LIN {X 0,Y 183.152,Z 369.76,A -85,B 0,C 180,E1 -22263.807,E2 -22263.807} C_VEL
LIN {X 0,Y 182.882,Z 372.565,A -85,B 0,C 180,E1 -22267.944,E2 -22267.944} C_VEL
LIN {X 0,Y 183.104,Z 373.609,A -85,B 0,C 180,E1 -22270.732,E2 -22270.732} C_VEL
LIN {X 0,Y 183.564,Z 374.058,A -85,B 0,C 180,E1 -22273.565,E2 -22273.565} C_VEL
LIN {X 0,Y 184.444,Z 373.742,A -85,B 0,C 180,E1 -22276.698,E2 -22276.698} C_VEL
LIN {X 0,Y 185.786,Z 372.532,A -85,B 0,C 180,E1 -22279.98,E2 -22279.98} C_VEL
LIN {X 0,Y 187.578,Z 370.431,A -85,B 0,C 180,E1 -22283.169,E2 -22283.169} C_VEL
LIN {X 0,Y 189.778,Z 367.45,A -85,B 0,C 180,E1 -22286.257,E2 -22286.257} C_VEL
LIN {X 0,Y 193.019,Z 362.657,A -85,B 0,C 180,E1 -22289.797,E2 -22289.797} C_VEL
LIN {X 0,Y 196.874,Z 356.364,A -85,B 0,C 180,E1 -22293.185,E2 -22293.185} C_VEL
LIN {X 0,Y 200.364,Z 350.078,A -85,B 0,C 180,E1 -22295.784,E2 -22295.784} C_VEL
LIN {X 0,Y 204.762,Z 341.315,A -85,B 0,C 180,E1 -22298.595,E2 -22298.595} C_VEL
LIN {X 0,Y 209.064,Z 331.687,A -85,B 0,C 180,E1 -22300.994,E2 -22300.994} C_VEL
LIN {X 0,Y 213.104,Z 321.145,A -85,B 0,C 180,E1 -22303.022,E2 -22303.022} C_VEL
LIN {X 0,Y 216.763,Z 309.855,A -85,B 0,C 180,E1 -22304.707,E2 -22304.707} C_VEL
LIN {X 0,Y 219.632,Z 298.789,A -85,B 0,C 180,E1 -22305.997,E2 -22305.997} C_VEL
LIN {X 0,Y 222.031,Z 286.626,A -85,B 0,C 180,E1 -22307.061,E2 -22307.061} C_VEL
LIN {X 0,Y 223.839,Z 274.15,A -85,B 0,C 180,E1 -22307.808,E2 -22307.808} C_VEL
LIN {X 0,Y 226.368,Z 244.862,A -85,B 0,C 180,E1 -22308.842,E2 -22308.842} C_VEL
LIN {X 0,Y 227.604,Z 229.196,A -85,B 0,C 180,E1 -22309.377,E2 -22309.377} C_VEL
LIN {X 0,Y 223.853,Z 221.057,A -85,B 0,C 180,E1 -22311.183,E2 -22311.183} C_VEL
LIN {X 0,Y 219.292,Z 213.106,A -85,B 0,C 180,E1 -22313.476,E2 -22313.476} C_VEL
LIN {X 0,Y 214.6,Z 205.629,A -85,B 0,C 180,E1 -22316.16,E2 -22316.16} C_VEL
LIN {X 0,Y 212.303,Z 202.347,A -85,B 0,C 180,E1 -22317.592,E2 -22317.592} C_VEL
LIN {X 0,Y 209.697,Z 198.642,A -85,B 0,C 180,E1 -22319.412,E2 -22319.412} C_VEL
LIN {X 0,Y 208.666,Z 197.162,A -85,B 0,C 180,E1 -22320.182,E2 -22320.182} C_VEL
LIN {X 0,Y 206.119,Z 193.314,A -85,B 0,C 180,E1 -22322.322,E2 -22322.322} C_VEL
LIN {X 0,Y 203.232,Z 190.633,A -85,B 0,C 180,E1 -22324.977,E2 -22324.977} C_VEL
LIN {X 0,Y 202.029,Z 188.256,A -85,B 0,C 180,E1 -22326.493,E2 -22326.493} C_VEL
LIN {X 0,Y 198.406,Z 185.102,A -85,B 0,C 180,E1 -22332.017,E2 -22332.017} C_VEL
LIN {X 0,Y 197.661,Z 183.274,A -85,B 0,C 180,E1 -22334.413,E2 -22334.413} C_VEL
LIN {X 0,Y 196.972,Z 183.268,A -85,B 0,C 180,E1 -22338.732,E2 -22338.732} C_VEL
LIN {X 0,Y 198.03,Z 184.97,A -85,B 0,C 180,E1 -22344.495,E2 -22344.495} C_VEL
LIN {X 0,Y 198.934,Z 186.56,A -85,B 0,C 180,E1 -22346.631,E2 -22346.631} C_VEL
LIN {X 0,Y 203.525,Z 193.122,A -85,B 0,C 180,E1 -22352.933,E2 -22352.933} C_VEL
LIN {X 0,Y 206.778,Z 198.314,A -85,B 0,C 180,E1 -22356.036,E2 -22356.036} C_VEL
LIN {X 0,Y 211.278,Z 205.799,A -85,B 0,C 180,E1 -22359.489,E2 -22359.489} C_VEL
LIN {X 0,Y 214.488,Z 211.478,A -85,B 0,C 180,E1 -22361.581,E2 -22361.581} C_VEL
LIN {X 0,Y 217.853,Z 217.949,A -85,B 0,C 180,E1 -22363.597,E2 -22363.597} C_VEL
LIN {X 0,Y 221.896,Z 226.386,A -85,B 0,C 180,E1 -22365.77,E2 -22365.77} C_VEL
LIN {X 0,Y 226.021,Z 237.025,A -85,B 0,C 180,E1 -22367.898,E2 -22367.898} C_VEL
LIN {X 0,Y 226.566,Z 244.834,A -85,B 0,C 180,E1 -22368.537,E2 -22368.537} C_VEL
LIN {X 0,Y 224.824,Z 267.129,A -85,B 0,C 180,E1 -22369.298,E2 -22369.298} C_VEL
LIN {X 0,Y 223.917,Z 272.973,A -85,B 0,C 180,E1 -22369.35,E2 -22369.35} C_VEL
LIN {X 0,Y 221.191,Z 282.484,A -85,B 0,C 180,E1 -22369.097,E2 -22369.097} C_VEL
LIN {X 0,Y 218.142,Z 291.897,A -85,B 0,C 180,E1 -22368.96,E2 -22368.96} C_VEL
LIN {X 0,Y 216.749,Z 297.576,A -85,B 0,C 180,E1 -22369.179,E2 -22369.179} C_VEL
LIN {X 0,Y 213.874,Z 310.256,A -85,B 0,C 180,E1 -22370.149,E2 -22370.149} C_VEL
LIN {X 0,Y 210.254,Z 322.7,A -85,B 0,C 180,E1 -22371.495,E2 -22371.495} C_VEL
LIN {X 0,Y 205.689,Z 335.169,A -85,B 0,C 180,E1 -22373.276,E2 -22373.276} C_VEL
LIN {X 0,Y 201.948,Z 344.09,A -85,B 0,C 180,E1 -22374.954,E2 -22374.954} C_VEL
LIN {X 0,Y 197.526,Z 353.357,A -85,B 0,C 180,E1 -22377.138,E2 -22377.138} C_VEL
LIN {X 0,Y 192.824,Z 362.381,A -85,B 0,C 180,E1 -22379.922,E2 -22379.922} C_VEL
LIN {X 0,Y 188.656,Z 369.747,A -85,B 0,C 180,E1 -22382.847,E2 -22382.847} C_VEL
LIN {X 0,Y 184.654,Z 376.594,A -85,B 0,C 180,E1 -22386.443,E2 -22386.443} C_VEL
LIN {X 0,Y 181.708,Z 381.181,A -85,B 0,C 180,E1 -22389.628,E2 -22389.628} C_VEL
LIN {X 0,Y 178.635,Z 385.659,A -85,B 0,C 180,E1 -22394.013,E2 -22394.013} C_VEL
LIN {X 0,Y 177.625,Z 387.289,A -85,B 0,C 180,E1 -22396.266,E2 -22396.266} C_VEL
LIN {X 0,Y 176.39,Z 389.3,A -85,B 0,C 180,E1 -22400.828,E2 -22400.828} C_VEL
LIN {X 0,Y 176.069,Z 389.772,A -85,B 0,C 180,E1 -22405.42,E2 -22405.42} C_VEL
LIN {X 0,Y 176.19,Z 389.418,A -85,B 0,C 180,E1 -22407.713,E2 -22407.713} C_VEL
LIN {X 0,Y 176.407,Z 388.626,A -85,B 0,C 180,E1 -22409.999,E2 -22409.999} C_VEL
LIN {X 0,Y 176.256,Z 387.392,A -85,B 0,C 180,E1 -22412.284,E2 -22412.284} C_VEL
LIN {X 0,Y 176.176,Z 384.702,A -85,B 0,C 180,E1 -22415.722,E2 -22415.722} C_VEL
LIN {X 0,Y 176.508,Z 380.942,A -85,B 0,C 180,E1 -22419.163,E2 -22419.163} C_VEL
LIN {X 0,Y 177.165,Z 375.989,A -85,B 0,C 180,E1 -22422.601,E2 -22422.601} C_VEL
LIN {X 0,Y 178.446,Z 369.723,A -85,B 0,C 180,E1 -22426.002,E2 -22426.002} C_VEL
LIN {X 0,Y 180.258,Z 361.863,A -85,B 0,C 180,E1 -22429.353,E2 -22429.353} C_VEL
LIN {X 0,Y 182.174,Z 353.728,A -85,B 0,C 180,E1 -22432.113,E2 -22432.113} C_VEL
LIN {X 0,Y 184.49,Z 343.939,A -85,B 0,C 180,E1 -22434.772,E2 -22434.772} C_VEL
LIN {X 0,Y 186.674,Z 334.322,A -85,B 0,C 180,E1 -22436.857,E2 -22436.857} C_VEL
LIN {X 0,Y 188.827,Z 324.044,A -85,B 0,C 180,E1 -22438.632,E2 -22438.632} C_VEL
LIN {X 0,Y 190.99,Z 311.886,A -85,B 0,C 180,E1 -22440.242,E2 -22440.242} C_VEL
LIN {X 0,Y 192.737,Z 299.331,A -85,B 0,C 180,E1 -22441.458,E2 -22441.458} C_VEL
LIN {X 0,Y 194.06,Z 286.706,A -85,B 0,C 180,E1 -22442.287,E2 -22442.287} C_VEL
LIN {X 0,Y 196.483,Z 238.495,A -85,B 0,C 180,E1 -22444.227,E2 -22444.227} C_VEL
LIN {X 0,Y 193.478,Z 211.936,A -85,B 0,C 180,E1 -22445.896,E2 -22445.896} C_VEL
LIN {X 0,Y 185.743,Z 191.175,A -85,B 0,C 180,E1 -22448.157,E2 -22448.157} C_VEL
LIN {X 0,Y 179.959,Z 177.42,A -85,B 0,C 180,E1 -22449.964,E2 -22449.964} C_VEL
LIN {X 0,Y 178.427,Z 171.263,A -85,B 0,C 180,E1 -22453.455,E2 -22453.455} C_VEL
LIN {X 0,Y 178.403,Z 171.26,A -85,B 0,C 180,E1 -22458.457,E2 -22458.457} C_VEL
LIN {X 0,Y 178.422,Z 171.263,A -85,B 0,C 180,E1 -22463.782,E2 -22463.782} C_VEL
LIN {X 0,Y 178.487,Z 171.252,A -85,B 0,C 180,E1 -22466.545,E2 -22466.545} C_VEL
LIN {X 0,Y 178.522,Z 171.241,A -85,B 0,C 180,E1 -22470.005,E2 -22470.005} C_VEL
LIN {X 0,Y 178.534,Z 171.244,A -85,B 0,C 180,E1 -22474.874,E2 -22474.874} C_VEL
LIN {X 0,Y 178.59,Z 171.24,A -85,B 0,C 180,E1 -22480.812,E2 -22480.812} C_VEL
LIN {X 0,Y 178.648,Z 171.23,A -85,B 0,C 180,E1 -22486.346,E2 -22486.346} C_VEL
LIN {X 0,Y 178.957,Z 171.183,A -85,B 0,C 180,E1 -22490.961,E2 -22490.961} C_VEL
LIN {X 0,Y 179.152,Z 171.167,A -85,B 0,C 180,E1 -22497.751,E2 -22497.751} C_VEL
LIN {X 0,Y 179.37,Z 171.135,A -85,B 0,C 180,E1 -22499.999,E2 -22499.999} C_VEL
LIN {X 0,Y 178.87,Z 171.194,A -85,B 0,C 180,E1 -22504.506,E2 -22504.506} C_VEL
LIN {X 0,Y 178.956,Z 171.192,A -85,B 0,C 180,E1 -22509.037,E2 -22509.037} C_VEL
LIN {X 0,Y 178.683,Z 171.207,A -85,B 0,C 180,E1 -22513.649,E2 -22513.649} C_VEL
LIN {X 0,Y 178.65,Z 171.229,A -85,B 0,C 180,E1 -22518.342,E2 -22518.342} C_VEL
LIN {X 0,Y 178.519,Z 171.237,A -85,B 0,C 180,E1 -22523.183,E2 -22523.183} C_VEL
LIN {X 0,Y 178.483,Z 171.241,A -85,B 0,C 180,E1 -22528.196,E2 -22528.196} C_VEL
LIN {X 0,Y 178.475,Z 171.249,A -85,B 0,C 180,E1 -22530.79,E2 -22530.79} C_VEL
LIN {X 0,Y 178.481,Z 171.24,A -85,B 0,C 180,E1 -22534.22,E2 -22534.22} C_VEL
LIN {X 0,Y 178.491,Z 171.243,A -85,B 0,C 180,E1 -22539.048,E2 -22539.048} C_VEL
LIN {X 0,Y 178.516,Z 171.246,A -85,B 0,C 180,E1 -22542.009,E2 -22542.009} C_VEL
LIN {X 0,Y 178.526,Z 171.235,A -85,B 0,C 180,E1 -22545.119,E2 -22545.119} C_VEL
LIN {X 0,Y 178.52,Z 171.244,A -85,B 0,C 180,E1 -22548.415,E2 -22548.415} C_VEL
LIN {X 0,Y 178.464,Z 171.245,A -85,B 0,C 180,E1 -22553.794,E2 -22553.794} C_VEL
LIN {X 0,Y 178.487,Z 171.249,A -85,B 0,C 180,E1 -22556.548,E2 -22556.548} C_VEL
LIN {X 0,Y 178.518,Z 171.246,A -85,B 0,C 180,E1 -22560.007,E2 -22560.007} C_VEL
LIN {X 0,Y 178.53,Z 171.246,A -85,B 0,C 180,E1 -22564.876,E2 -22564.876} C_VEL
LIN {X 0,Y 178.619,Z 171.236,A -85,B 0,C 180,E1 -22570.785,E2 -22570.785} C_VEL
LIN {X 0,Y 178.662,Z 171.232,A -85,B 0,C 180,E1 -22574.018,E2 -22574.018} C_VEL
LIN {X 0,Y 178.891,Z 171.207,A -85,B 0,C 180,E1 -22579.155,E2 -22579.155} C_VEL
LIN {X 0,Y 178.931,Z 171.202,A -85,B 0,C 180,E1 -22583.234,E2 -22583.234} C_VEL
LIN {X 0,Y 179.216,Z 171.163,A -85,B 0,C 180,E1 -22588.449,E2 -22588.449} C_VEL
LIN {X 0,Y 180.365,Z 174.204,A -85,B 0,C 180,E1 -22588.849,E2 -22588.849} C_VEL
LIN {X 0,Y 182.731,Z 178.435,A -85,B 0,C 180,E1 -22589.501,E2 -22589.501} C_VEL
LIN {X 0,Y 193.933,Z 202.509,A -85,B 0,C 180,E1 -22592.563,E2 -22592.563} C_VEL
LIN {X 0,Y 197.479,Z 211.708,A -85,B 0,C 180,E1 -22593.518,E2 -22593.518} C_VEL
LIN {X 0,Y 194.431,Z 270.668,A -85,B 0,C 180,E1 -22595.874,E2 -22595.874} C_VEL
LIN {X 0,Y 193.172,Z 283.987,A -85,B 0,C 180,E1 -22596.792,E2 -22596.792} C_VEL
LIN {X 0,Y 191.66,Z 296.7,A -85,B 0,C 180,E1 -22598.093,E2 -22598.093} C_VEL
LIN {X 0,Y 189.618,Z 309.391,A -85,B 0,C 180,E1 -22599.872,E2 -22599.872} C_VEL
LIN {X 0,Y 187.503,Z 319.771,A -85,B 0,C 180,E1 -22601.731,E2 -22601.731} C_VEL
LIN {X 0,Y 185.281,Z 329.824,A -85,B 0,C 180,E1 -22603.995,E2 -22603.995} C_VEL
LIN {X 0,Y 183.062,Z 339.34,A -85,B 0,C 180,E1 -22606.7,E2 -22606.7} C_VEL
LIN {X 0,Y 180.889,Z 348.221,A -85,B 0,C 180,E1 -22609.876,E2 -22609.876} C_VEL
LIN {X 0,Y 179.194,Z 355.371,A -85,B 0,C 180,E1 -22613.093,E2 -22613.093} C_VEL
LIN {X 0,Y 177.843,Z 361.2,A -85,B 0,C 180,E1 -22616.398,E2 -22616.398} C_VEL
LIN {X 0,Y 176.795,Z 366.194,A -85,B 0,C 180,E1 -22620.069,E2 -22620.069} C_VEL
LIN {X 0,Y 176.043,Z 370.093,A -85,B 0,C 180,E1 -22623.982,E2 -22623.982} C_VEL
LIN {X 0,Y 175.806,Z 372.183,A -85,B 0,C 180,E1 -22626.918,E2 -22626.918} C_VEL
LIN {X 0,Y 176.006,Z 373.819,A -85,B 0,C 180,E1 -22630.654,E2 -22630.654} C_VEL
LIN {X 0,Y 176.634,Z 374.398,A -85,B 0,C 180,E1 -22634.261,E2 -22634.261} C_VEL
LIN {X 0,Y 178.019,Z 373.758,A -85,B 0,C 180,E1 -22638.601,E2 -22638.601} C_VEL
LIN {X 0,Y 179.473,Z 372.502,A -85,B 0,C 180,E1 -22641.555,E2 -22641.555} C_VEL
LIN {X 0,Y 182.319,Z 369.171,A -85,B 0,C 180,E1 -22645.976,E2 -22645.976} C_VEL
LIN {X 0,Y 184.763,Z 365.948,A -85,B 0,C 180,E1 -22648.858,E2 -22648.858} C_VEL
LIN {X 0,Y 188.498,Z 360.566,A -85,B 0,C 180,E1 -22652.412,E2 -22652.412} C_VEL
LIN {X 0,Y 192.735,Z 353.781,A -85,B 0,C 180,E1 -22655.732,E2 -22655.732} C_VEL
LIN {X 0,Y 197.393,Z 345.494,A -85,B 0,C 180,E1 -22658.776,E2 -22658.776} C_VEL
LIN {X 0,Y 201.87,Z 336.52,A -85,B 0,C 180,E1 -22661.319,E2 -22661.319} C_VEL
LIN {X 0,Y 206.159,Z 326.687,A -85,B 0,C 180,E1 -22663.463,E2 -22663.463} C_VEL
LIN {X 0,Y 210.089,Z 315.911,A -85,B 0,C 180,E1 -22665.315,E2 -22665.315} C_VEL
LIN {X 0,Y 213.712,Z 304.033,A -85,B 0,C 180,E1 -22666.877,E2 -22666.877} C_VEL
LIN {X 0,Y 216.674,Z 291.098,A -85,B 0,C 180,E1 -22668.153,E2 -22668.153} C_VEL
LIN {X 0,Y 218.974,Z 277.674,A -85,B 0,C 180,E1 -22669.072,E2 -22669.072} C_VEL
LIN {X 0,Y 220.63,Z 261.781,A -85,B 0,C 180,E1 -22669.716,E2 -22669.716} C_VEL
LIN {X 0,Y 223.109,Z 232.103,A -85,B 0,C 180,E1 -22670.735,E2 -22670.735} C_VEL
LIN {X 0,Y 220.246,Z 225.744,A -85,B 0,C 180,E1 -22672.22,E2 -22672.22} C_VEL
LIN {X 0,Y 216.072,Z 218.258,A -85,B 0,C 180,E1 -22674.489,E2 -22674.489} C_VEL
LIN {X 0,Y 212.079,Z 211.691,A -85,B 0,C 180,E1 -22676.904,E2 -22676.904} C_VEL
LIN {X 0,Y 209.888,Z 208.452,A -85,B 0,C 180,E1 -22678.382,E2 -22678.382} C_VEL
LIN {X 0,Y 206.592,Z 203.502,A -85,B 0,C 180,E1 -22680.858,E2 -22680.858} C_VEL
LIN {X 0,Y 204.299,Z 199.922,A -85,B 0,C 180,E1 -22682.916,E2 -22682.916} C_VEL
LIN {X 0,Y 201.545,Z 197.137,A -85,B 0,C 180,E1 -22685.612,E2 -22685.612} C_VEL
LIN {X 0,Y 200.472,Z 195.04,A -85,B 0,C 180,E1 -22687.049,E2 -22687.049} C_VEL
LIN {X 0,Y 197.009,Z 191.646,A -85,B 0,C 180,E1 -22692.884,E2 -22692.884} C_VEL
LIN {X 0,Y 196.459,Z 190.222,A -85,B 0,C 180,E1 -22695.005,E2 -22695.005} C_VEL
LIN {X 0,Y 195.945,Z 190.417,A -85,B 0,C 180,E1 -22699.378,E2 -22699.378} C_VEL
LIN {X 0,Y 196.964,Z 192.038,A -85,B 0,C 180,E1 -22704.458,E2 -22704.458} C_VEL
LIN {X 0,Y 197.731,Z 193.544,A -85,B 0,C 180,E1 -22706.379,E2 -22706.379} C_VEL
LIN {X 0,Y 201.882,Z 199.809,A -85,B 0,C 180,E1 -22712.403,E2 -22712.403} C_VEL
LIN {X 0,Y 204.836,Z 204.736,A -85,B 0,C 180,E1 -22715.386,E2 -22715.386} C_VEL
LIN {X 0,Y 208.902,Z 211.858,A -85,B 0,C 180,E1 -22718.701,E2 -22718.701} C_VEL
LIN {X 0,Y 211.931,Z 217.566,A -85,B 0,C 180,E1 -22720.832,E2 -22720.832} C_VEL
LIN {X 0,Y 215.483,Z 224.666,A -85,B 0,C 180,E1 -22723.061,E2 -22723.061} C_VEL
LIN {X 0,Y 218.978,Z 232.69,A -85,B 0,C 180,E1 -22725.082,E2 -22725.082} C_VEL
LIN {X 0,Y 221.903,Z 240.663,A -85,B 0,C 180,E1 -22726.706,E2 -22726.706} C_VEL
LIN {X 0,Y 222.119,Z 246.606,A -85,B 0,C 180,E1 -22727.166,E2 -22727.166} C_VEL
LIN {X 0,Y 218.697,Z 285.548,A -85,B 0,C 180,E1 -22728.538,E2 -22728.538} C_VEL
LIN {X 0,Y 216.749,Z 297.576,A -85,B 0,C 180,E1 -22729.179,E2 -22729.179} C_VEL
LIN {X 0,Y 215.143,Z 303.212,A -85,B 0,C 180,E1 -22729.428,E2 -22729.428} C_VEL
LIN {X 0,Y 211.028,Z 312.255,A -85,B 0,C 180,E1 -22729.621,E2 -22729.621} C_VEL
LIN {X 0,Y 206.531,Z 320.965,A -85,B 0,C 180,E1 -22729.951,E2 -22729.951} C_VEL
LIN {X 0,Y 204.316,Z 326.046,A -85,B 0,C 180,E1 -22730.459,E2 -22730.459} C_VEL
LIN {X 0,Y 199.597,Z 337.708,A -85,B 0,C 180,E1 -22732.279,E2 -22732.279} C_VEL
LIN {X 0,Y 195.306,Z 347.133,A -85,B 0,C 180,E1 -22734.213,E2 -22734.213} C_VEL
LIN {X 0,Y 190.884,Z 355.805,A -85,B 0,C 180,E1 -22736.475,E2 -22736.475} C_VEL
LIN {X 0,Y 185.988,Z 364.333,A -85,B 0,C 180,E1 -22739.326,E2 -22739.326} C_VEL
LIN {X 0,Y 181.738,Z 371.226,A -85,B 0,C 180,E1 -22742.35,E2 -22742.35} C_VEL
LIN {X 0,Y 178.175,Z 376.803,A -85,B 0,C 180,E1 -22745.532,E2 -22745.532} C_VEL
LIN {X 0,Y 175.037,Z 381.262,A -85,B 0,C 180,E1 -22748.815,E2 -22748.815} C_VEL
LIN {X 0,Y 173.316,Z 383.653,A -85,B 0,C 180,E1 -22751.069,E2 -22751.069} C_VEL
LIN {X 0,Y 171.806,Z 385.628,A -85,B 0,C 180,E1 -22753.359,E2 -22753.359} C_VEL
LIN {X 0,Y 170.691,Z 387.166,A -85,B 0,C 180,E1 -22755.696,E2 -22755.696} C_VEL
LIN {X 0,Y 169.355,Z 389.046,A -85,B 0,C 180,E1 -22760.444,E2 -22760.444} C_VEL
LIN {X 0,Y 168.999,Z 389.41,A -85,B 0,C 180,E1 -22765.228,E2 -22765.228} C_VEL
LIN {X 0,Y 169.108,Z 388.967,A -85,B 0,C 180,E1 -22767.617,E2 -22767.617} C_VEL
LIN {X 0,Y 169.342,Z 388.127,A -85,B 0,C 180,E1 -22769.999,E2 -22769.999} C_VEL
LIN {X 0,Y 169.108,Z 385.625,A -85,B 0,C 180,E1 -22774.101,E2 -22774.101} C_VEL
LIN {X 0,Y 169.33,Z 381.61,A -85,B 0,C 180,E1 -22778.351,E2 -22778.351} C_VEL
LIN {X 0,Y 169.908,Z 376.938,A -85,B 0,C 180,E1 -22781.935,E2 -22781.935} C_VEL
LIN {X 0,Y 171.047,Z 370.964,A -85,B 0,C 180,E1 -22785.489,E2 -22785.489} C_VEL
LIN {X 0,Y 172.773,Z 363.48,A -85,B 0,C 180,E1 -22788.99,E2 -22788.99} C_VEL
LIN {X 0,Y 174.69,Z 355.266,A -85,B 0,C 180,E1 -22792.052,E2 -22792.052} C_VEL
LIN {X 0,Y 176.995,Z 346.576,A -85,B 0,C 180,E1 -22794.639,E2 -22794.639} C_VEL
LIN {X 0,Y 179.5,Z 336.296,A -85,B 0,C 180,E1 -22797.074,E2 -22797.074} C_VEL
LIN {X 0,Y 181.589,Z 326.481,A -85,B 0,C 180,E1 -22798.931,E2 -22798.931} C_VEL
LIN {X 0,Y 183.935,Z 314.161,A -85,B 0,C 180,E1 -22800.732,E2 -22800.732} C_VEL
LIN {X 0,Y 185.744,Z 302.626,A -85,B 0,C 180,E1 -22801.985,E2 -22801.985} C_VEL
LIN {X 0,Y 187.274,Z 289.551,A -85,B 0,C 180,E1 -22802.965,E2 -22802.965} C_VEL
LIN {X 0,Y 188.434,Z 271.783,A -85,B 0,C 180,E1 -22803.775,E2 -22803.775} C_VEL
LIN {X 0,Y 189.991,Z 238.867,A -85,B 0,C 180,E1 -22805.129,E2 -22805.129} C_VEL
LIN {X 0,Y 187.411,Z 214.466,A -85,B 0,C 180,E1 -22806.713,E2 -22806.713} C_VEL
LIN {X 0,Y 180.168,Z 194.799,A -85,B 0,C 180,E1 -22808.952,E2 -22808.952} C_VEL
LIN {X 0,Y 173.988,Z 180.443,A -85,B 0,C 180,E1 -22810.881,E2 -22810.881} C_VEL
LIN {X 0,Y 172.549,Z 177.061,A -85,B 0,C 180,E1 -22811.419,E2 -22811.419} C_VEL
LIN {X 0,Y 171.374,Z 172.141,A -85,B 0,C 180,E1 -22814.391,E2 -22814.391} C_VEL
LIN {X 0,Y 171.335,Z 172.141,A -85,B 0,C 180,E1 -22818.98,E2 -22818.98} C_VEL
LIN {X 0,Y 171.387,Z 172.136,A -85,B 0,C 180,E1 -22822.039,E2 -22822.039} C_VEL
LIN {X 0,Y 171.398,Z 172.134,A -85,B 0,C 180,E1 -22825.091,E2 -22825.091} C_VEL
LIN {X 0,Y 171.449,Z 172.121,A -85,B 0,C 180,E1 -22830.533,E2 -22830.533} C_VEL
LIN {X 0,Y 171.455,Z 172.119,A -85,B 0,C 180,E1 -22835.8,E2 -22835.8} C_VEL
LIN {X 0,Y 171.546,Z 172.117,A -85,B 0,C 180,E1 -22840.866,E2 -22840.866} C_VEL
LIN {X 0,Y 171.561,Z 172.113,A -85,B 0,C 180,E1 -22845.77,E2 -22845.77} C_VEL
LIN {X 0,Y 171.886,Z 172.066,A -85,B 0,C 180,E1 -22850.586,E2 -22850.586} C_VEL
LIN {X 0,Y 171.821,Z 172.08,A -85,B 0,C 180,E1 -22855.306,E2 -22855.306} C_VEL
LIN {X 0,Y 172.333,Z 172.012,A -85,B 0,C 180,E1 -22859.999,E2 -22859.999} C_VEL
LIN {X 0,Y 171.819,Z 172.073,A -85,B 0,C 180,E1 -22864.691,E2 -22864.691} C_VEL
LIN {X 0,Y 171.885,Z 172.071,A -85,B 0,C 180,E1 -22869.412,E2 -22869.412} C_VEL
LIN {X 0,Y 171.606,Z 172.088,A -85,B 0,C 180,E1 -22874.223,E2 -22874.223} C_VEL
LIN {X 0,Y 171.542,Z 172.114,A -85,B 0,C 180,E1 -22879.563,E2 -22879.563} C_VEL
LIN {X 0,Y 171.465,Z 172.101,A -85,B 0,C 180,E1 -22885.616,E2 -22885.616} C_VEL
LIN {X 0,Y 171.437,Z 172.126,A -85,B 0,C 180,E1 -22890.586,E2 -22890.586} C_VEL
LIN {X 0,Y 171.404,Z 172.118,A -85,B 0,C 180,E1 -22895.03,E2 -22895.03} C_VEL
LIN {X 0,Y 171.443,Z 172.121,A -85,B 0,C 180,E1 -22898.845,E2 -22898.845} C_VEL
LIN {X 0,Y 171.45,Z 172.118,A -85,B 0,C 180,E1 -22904.173,E2 -22904.173} C_VEL
LIN {X 0,Y 171.436,Z 172.126,A -85,B 0,C 180,E1 -22909.013,E2 -22909.013} C_VEL
LIN {X 0,Y 171.44,Z 172.126,A -85,B 0,C 180,E1 -22912.056,E2 -22912.056} C_VEL
LIN {X 0,Y 171.423,Z 172.132,A -85,B 0,C 180,E1 -22917.795,E2 -22917.795} C_VEL
LIN {X 0,Y 171.445,Z 172.127,A -85,B 0,C 180,E1 -22920.535,E2 -22920.535} C_VEL
LIN {X 0,Y 171.453,Z 172.128,A -85,B 0,C 180,E1 -22925.802,E2 -22925.802} C_VEL
LIN {X 0,Y 171.575,Z 172.114,A -85,B 0,C 180,E1 -22930.873,E2 -22930.873} C_VEL
LIN {X 0,Y 171.606,Z 172.113,A -85,B 0,C 180,E1 -22935.777,E2 -22935.777} C_VEL
LIN {X 0,Y 171.907,Z 172.075,A -85,B 0,C 180,E1 -22940.589,E2 -22940.589} C_VEL
LIN {X 0,Y 171.932,Z 172.07,A -85,B 0,C 180,E1 -22946.486,E2 -22946.486} C_VEL
LIN {X 0,Y 171.994,Z 172.064,A -85,B 0,C 180,E1 -22947.074,E2 -22947.074} C_VEL
LIN {X 0,Y 173.209,Z 175.119,A -85,B 0,C 180,E1 -22947.519,E2 -22947.519} C_VEL
LIN {X 0,Y 174.549,Z 177.336,A -85,B 0,C 180,E1 -22947.91,E2 -22947.91} C_VEL
LIN {X 0,Y 177.741,Z 183.259,A -85,B 0,C 180,E1 -22948.845,E2 -22948.845} C_VEL
LIN {X 0,Y 188.037,Z 205.509,A -85,B 0,C 180,E1 -22951.78,E2 -22951.78} C_VEL
LIN {X 0,Y 191.175,Z 213.616,A -85,B 0,C 180,E1 -22952.671,E2 -22952.671} C_VEL
LIN {X 0,Y 187.931,Z 271.256,A -85,B 0,C 180,E1 -22955.03,E2 -22955.03} C_VEL
LIN {X 0,Y 186.653,Z 284.156,A -85,B 0,C 180,E1 -22955.945,E2 -22955.945} C_VEL
LIN {X 0,Y 185.227,Z 295.864,A -85,B 0,C 180,E1 -22957.162,E2 -22957.162} C_VEL
LIN {X 0,Y 183.28,Z 307.849,A -85,B 0,C 180,E1 -22958.824,E2 -22958.824} C_VEL
LIN {X 0,Y 180.924,Z 319.414,A -85,B 0,C 180,E1 -22960.917,E2 -22960.917} C_VEL
LIN {X 0,Y 178.571,Z 329.585,A -85,B 0,C 180,E1 -22963.252,E2 -22963.252} C_VEL
LIN {X 0,Y 176.641,Z 337.742,A -85,B 0,C 180,E1 -22965.58,E2 -22965.58} C_VEL
LIN {X 0,Y 174.303,Z 346.914,A -85,B 0,C 180,E1 -22968.82,E2 -22968.82} C_VEL
LIN {X 0,Y 172.484,Z 354.33,A -85,B 0,C 180,E1 -22972.143,E2 -22972.143} C_VEL
LIN {X 0,Y 170.814,Z 361.212,A -85,B 0,C 180,E1 -22976.068,E2 -22976.068} C_VEL
LIN {X 0,Y 169.742,Z 366.195,A -85,B 0,C 180,E1 -22979.793,E2 -22979.793} C_VEL
LIN {X 0,Y 168.985,Z 370.071,A -85,B 0,C 180,E1 -22983.72,E2 -22983.72} C_VEL
LIN {X 0,Y 168.716,Z 372.739,A -85,B 0,C 180,E1 -22987.68,E2 -22987.68} C_VEL
LIN {X 0,Y 169.027,Z 374.29,A -85,B 0,C 180,E1 -22991.705,E2 -22991.705} C_VEL
LIN {X 0,Y 169.77,Z 374.731,A -85,B 0,C 180,E1 -22995.273,E2 -22995.273} C_VEL
LIN {X 0,Y 171.021,Z 374.266,A -85,B 0,C 180,E1 -22998.892,E2 -22998.892} C_VEL
LIN {X 0,Y 172.757,Z 372.905,A -85,B 0,C 180,E1 -23002.396,E2 -23002.396} C_VEL
LIN {X 0,Y 174.923,Z 370.66,A -85,B 0,C 180,E1 -23005.774,E2 -23005.774} C_VEL
LIN {X 0,Y 178.525,Z 366.329,A -85,B 0,C 180,E1 -23010.008,E2 -23010.008} C_VEL
LIN {X 0,Y 181.612,Z 362.266,A -85,B 0,C 180,E1 -23012.882,E2 -23012.882} C_VEL
LIN {X 0,Y 185.958,Z 355.862,A -85,B 0,C 180,E1 -23016.314,E2 -23016.314} C_VEL
LIN {X 0,Y 190.089,Z 349.267,A -85,B 0,C 180,E1 -23018.998,E2 -23018.998} C_VEL
LIN {X 0,Y 195.035,Z 340.205,A -85,B 0,C 180,E1 -23021.884,E2 -23021.884} C_VEL
LIN {X 0,Y 199.859,Z 330.148,A -85,B 0,C 180,E1 -23024.289,E2 -23024.289} C_VEL
LIN {X 0,Y 204.413,Z 319.023,A -85,B 0,C 180,E1 -23026.357,E2 -23026.357} C_VEL
LIN {X 0,Y 208.353,Z 307.207,A -85,B 0,C 180,E1 -23028.022,E2 -23028.022} C_VEL
LIN {X 0,Y 211.513,Z 295.152,A -85,B 0,C 180,E1 -23029.323,E2 -23029.323} C_VEL
LIN {X 0,Y 213.983,Z 282.58,A -85,B 0,C 180,E1 -23030.301,E2 -23030.301} C_VEL
LIN {X 0,Y 215.773,Z 269.599,A -85,B 0,C 180,E1 -23030.934,E2 -23030.934} C_VEL
LIN {X 0,Y 218.77,Z 234.856,A -85,B 0,C 180,E1 -23032.167,E2 -23032.167} C_VEL
LIN {X 0,Y 215.343,Z 227.777,A -85,B 0,C 180,E1 -23034.087,E2 -23034.087} C_VEL
LIN {X 0,Y 210.79,Z 219.668,A -85,B 0,C 180,E1 -23036.88,E2 -23036.88} C_VEL
LIN {X 0,Y 207.695,Z 214.73,A -85,B 0,C 180,E1 -23039.061,E2 -23039.061} C_VEL
LIN {X 0,Y 204.418,Z 209.594,A -85,B 0,C 180,E1 -23041.698,E2 -23041.698} C_VEL
LIN {X 0,Y 202.52,Z 206.526,A -85,B 0,C 180,E1 -23043.506,E2 -23043.506} C_VEL
LIN {X 0,Y 199.968,Z 203.786,A -85,B 0,C 180,E1 -23046.172,E2 -23046.172} C_VEL
LIN {X 0,Y 198.936,Z 201.829,A -85,B 0,C 180,E1 -23047.614,E2 -23047.614} C_VEL
LIN {X 0,Y 195.751,Z 198.339,A -85,B 0,C 180,E1 -23053.497,E2 -23053.497} C_VEL
LIN {X 0,Y 195.422,Z 197.245,A -85,B 0,C 180,E1 -23054.999,E2 -23054.999} C_VEL
LIN {X 0,Y 194.91,Z 197.456,A -85,B 0,C 180,E1 -23059.485,E2 -23059.485} C_VEL
LIN {X 0,Y 195.864,Z 199.078,A -85,B 0,C 180,E1 -23064.336,E2 -23064.336} C_VEL
LIN {X 0,Y 196.958,Z 201.495,A -85,B 0,C 180,E1 -23067.063,E2 -23067.063} C_VEL
LIN {X 0,Y 200.184,Z 206.369,A -85,B 0,C 180,E1 -23071.778,E2 -23071.778} C_VEL
LIN {X 0,Y 203.446,Z 212.2,A -85,B 0,C 180,E1 -23075.223,E2 -23075.223} C_VEL
LIN {X 0,Y 206.699,Z 218.202,A -85,B 0,C 180,E1 -23078.002,E2 -23078.002} C_VEL
LIN {X 0,Y 209.162,Z 223.084,A -85,B 0,C 180,E1 -23079.878,E2 -23079.878} C_VEL
LIN {X 0,Y 212.366,Z 229.737,A -85,B 0,C 180,E1 -23082.029,E2 -23082.029} C_VEL
LIN {X 0,Y 215.482,Z 237.33,A -85,B 0,C 180,E1 -23084.012,E2 -23084.012} C_VEL
LIN {X 0,Y 217.813,Z 243.805,A -85,B 0,C 180,E1 -23085.39,E2 -23085.39} C_VEL
LIN {X 0,Y 217.984,Z 246.943,A -85,B 0,C 180,E1 -23085.668,E2 -23085.668} C_VEL
LIN {X 0,Y 214.452,Z 285.28,A -85,B 0,C 180,E1 -23087.028,E2 -23087.028} C_VEL
LIN {X 0,Y 212.123,Z 298.724,A -85,B 0,C 180,E1 -23087.761,E2 -23087.761} C_VEL
LIN {X 0,Y 209.126,Z 310.982,A -85,B 0,C 180,E1 -23088.734,E2 -23088.734} C_VEL
LIN {X 0,Y 205.361,Z 323.105,A -85,B 0,C 180,E1 -23090.082,E2 -23090.082} C_VEL
LIN {X 0,Y 204.316,Z 326.046,A -85,B 0,C 180,E1 -23090.459,E2 -23090.459} C_VEL
LIN {X 0,Y 201.99,Z 331.076,A -85,B 0,C 180,E1 -23091.038,E2 -23091.038} C_VEL
LIN {X 0,Y 194.337,Z 342.069,A -85,B 0,C 180,E1 -23092.103,E2 -23092.103} C_VEL
LIN {X 0,Y 190.002,Z 348.007,A -85,B 0,C 180,E1 -23092.981,E2 -23092.981} C_VEL
LIN {X 0,Y 188.25,Z 350.791,A -85,B 0,C 180,E1 -23093.607,E2 -23093.607} C_VEL
LIN {X 0,Y 183.318,Z 359.576,A -85,B 0,C 180,E1 -23096.226,E2 -23096.226} C_VEL
LIN {X 0,Y 178.403,Z 367.315,A -85,B 0,C 180,E1 -23099.193,E2 -23099.193} C_VEL
LIN {X 0,Y 174.157,Z 373.583,A -85,B 0,C 180,E1 -23102.349,E2 -23102.349} C_VEL
LIN {X 0,Y 170.55,Z 378.624,A -85,B 0,C 180,E1 -23105.663,E2 -23105.663} C_VEL
LIN {X 0,Y 167.512,Z 382.586,A -85,B 0,C 180,E1 -23109.106,E2 -23109.106} C_VEL
LIN {X 0,Y 165.005,Z 385.567,A -85,B 0,C 180,E1 -23112.652,E2 -23112.652} C_VEL
LIN {X 0,Y 162.927,Z 388.099,A -85,B 0,C 180,E1 -23117.543,E2 -23117.543} C_VEL
LIN {X 0,Y 161.984,Z 389.109,A -85,B 0,C 180,E1 -23122.52,E2 -23122.52} C_VEL
LIN {X 0,Y 161.941,Z 388.766,A -85,B 0,C 180,E1 -23126.548,E2 -23126.548} C_VEL
LIN {X 0,Y 162.278,Z 387.619,A -85,B 0,C 180,E1 -23129.999,E2 -23129.999} C_VEL
LIN {X 0,Y 162.027,Z 385.27,A -85,B 0,C 180,E1 -23133.922,E2 -23133.922} C_VEL
LIN {X 0,Y 162.146,Z 382.161,A -85,B 0,C 180,E1 -23137.47,E2 -23137.47} C_VEL
LIN {X 0,Y 162.654,Z 377.776,A -85,B 0,C 180,E1 -23141.21,E2 -23141.21} C_VEL
LIN {X 0,Y 163.631,Z 372.131,A -85,B 0,C 180,E1 -23144.932,E2 -23144.932} C_VEL
LIN {X 0,Y 165.385,Z 365.063,A -85,B 0,C 180,E1 -23148.583,E2 -23148.583} C_VEL
LIN {X 0,Y 167.13,Z 357.781,A -85,B 0,C 180,E1 -23151.588,E2 -23151.588} C_VEL
LIN {X 0,Y 169.475,Z 348.976,A -85,B 0,C 180,E1 -23154.498,E2 -23154.498} C_VEL
LIN {X 0,Y 172.265,Z 338.155,A -85,B 0,C 180,E1 -23157.319,E2 -23157.319} C_VEL
LIN {X 0,Y 174.379,Z 328.812,A -85,B 0,C 180,E1 -23159.252,E2 -23159.252} C_VEL
LIN {X 0,Y 176.751,Z 317.279,A -85,B 0,C 180,E1 -23161.123,E2 -23161.123} C_VEL
LIN {X 0,Y 178.991,Z 304.226,A -85,B 0,C 180,E1 -23162.674,E2 -23162.674} C_VEL
LIN {X 0,Y 180.605,Z 291.289,A -85,B 0,C 180,E1 -23163.76,E2 -23163.76} C_VEL
LIN {X 0,Y 181.774,Z 276.222,A -85,B 0,C 180,E1 -23164.516,E2 -23164.516} C_VEL
LIN {X 0,Y 183.642,Z 239.785,A -85,B 0,C 180,E1 -23166.053,E2 -23166.053} C_VEL
LIN {X 0,Y 181.288,Z 216.656,A -85,B 0,C 180,E1 -23167.619,E2 -23167.619} C_VEL
LIN {X 0,Y 173.851,Z 196.488,A -85,B 0,C 180,E1 -23170.02,E2 -23170.02} C_VEL
LIN {X 0,Y 168.394,Z 183.893,A -85,B 0,C 180,E1 -23171.825,E2 -23171.825} C_VEL
LIN {X 0,Y 165.198,Z 176.747,A -85,B 0,C 180,E1 -23172.975,E2 -23172.975} C_VEL
LIN {X 0,Y 164.309,Z 173.02,A -85,B 0,C 180,E1 -23175.325,E2 -23175.325} C_VEL
LIN {X 0,Y 164.295,Z 173.02,A -85,B 0,C 180,E1 -23180.35,E2 -23180.35} C_VEL
LIN {X 0,Y 164.329,Z 173.015,A -85,B 0,C 180,E1 -23186.22,E2 -23186.22} C_VEL
LIN {X 0,Y 164.405,Z 173.004,A -85,B 0,C 180,E1 -23189.136,E2 -23189.136} C_VEL
LIN {X 0,Y 164.415,Z 173.003,A -85,B 0,C 180,E1 -23194.692,E2 -23194.692} C_VEL
LIN {X 0,Y 164.442,Z 173.001,A -85,B 0,C 180,E1 -23200.089,E2 -23200.089} C_VEL
LIN {X 0,Y 164.488,Z 172.989,A -85,B 0,C 180,E1 -23205.145,E2 -23205.145} C_VEL
LIN {X 0,Y 164.8,Z 172.952,A -85,B 0,C 180,E1 -23210.177,E2 -23210.177} C_VEL
LIN {X 0,Y 164.849,Z 172.935,A -85,B 0,C 180,E1 -23212.65,E2 -23212.65} C_VEL
LIN {X 0,Y 165.048,Z 172.924,A -85,B 0,C 180,E1 -23217.558,E2 -23217.558} C_VEL
LIN {X 0,Y 165.295,Z 172.888,A -85,B 0,C 180,E1 -23219.999,E2 -23219.999} C_VEL
LIN {X 0,Y 164.824,Z 172.95,A -85,B 0,C 180,E1 -23227.072,E2 -23227.072} C_VEL
LIN {X 0,Y 164.75,Z 172.954,A -85,B 0,C 180,E1 -23231.151,E2 -23231.151} C_VEL
LIN {X 0,Y 164.505,Z 172.988,A -85,B 0,C 180,E1 -23237.399,E2 -23237.399} C_VEL
LIN {X 0,Y 164.47,Z 172.996,A -85,B 0,C 180,E1 -23239.988,E2 -23239.988} C_VEL
LIN {X 0,Y 164.389,Z 172.983,A -85,B 0,C 180,E1 -23246.133,E2 -23246.133} C_VEL
LIN {X 0,Y 164.372,Z 173.005,A -85,B 0,C 180,E1 -23251.228,E2 -23251.228} C_VEL
LIN {X 0,Y 164.348,Z 172.992,A -85,B 0,C 180,E1 -23256.774,E2 -23256.774} C_VEL
LIN {X 0,Y 164.375,Z 173.003,A -85,B 0,C 180,E1 -23259.89,E2 -23259.89} C_VEL
LIN {X 0,Y 164.39,Z 173.003,A -85,B 0,C 180,E1 -23263.384,E2 -23263.384} C_VEL
LIN {X 0,Y 164.394,Z 172.993,A -85,B 0,C 180,E1 -23266.844,E2 -23266.844} C_VEL
LIN {X 0,Y 164.376,Z 173.009,A -85,B 0,C 180,E1 -23270.316,E2 -23270.316} C_VEL
LIN {X 0,Y 164.344,Z 173.001,A -85,B 0,C 180,E1 -23274.34,E2 -23274.34} C_VEL
LIN {X 0,Y 164.401,Z 173.007,A -85,B 0,C 180,E1 -23279.138,E2 -23279.138} C_VEL
LIN {X 0,Y 164.412,Z 173.004,A -85,B 0,C 180,E1 -23284.695,E2 -23284.695} C_VEL
LIN {X 0,Y 164.48,Z 172.997,A -85,B 0,C 180,E1 -23290.052,E2 -23290.052} C_VEL
LIN {X 0,Y 164.549,Z 172.99,A -85,B 0,C 180,E1 -23295.153,E2 -23295.153} C_VEL
LIN {X 0,Y 164.849,Z 172.954,A -85,B 0,C 180,E1 -23300.183,E2 -23300.183} C_VEL
LIN {X 0,Y 164.774,Z 172.965,A -85,B 0,C 180,E1 -23305.108,E2 -23305.108} C_VEL
LIN {X 0,Y 164.802,Z 172.959,A -85,B 0,C 180,E1 -23305.568,E2 -23305.568} C_VEL
LIN {X 0,Y 165.879,Z 175.875,A -85,B 0,C 180,E1 -23306.017,E2 -23306.017} C_VEL
LIN {X 0,Y 167.484,Z 178.323,A -85,B 0,C 180,E1 -23306.509,E2 -23306.509} C_VEL
LIN {X 0,Y 172.106,Z 186.58,A -85,B 0,C 180,E1 -23307.938,E2 -23307.938} C_VEL
LIN {X 0,Y 182.317,Z 208.87,A -85,B 0,C 180,E1 -23310.993,E2 -23310.993} C_VEL
LIN {X 0,Y 184.807,Z 215.595,A -85,B 0,C 180,E1 -23311.754,E2 -23311.754} C_VEL
LIN {X 0,Y 181.535,Z 271,A -85,B 0,C 180,E1 -23314.073,E2 -23314.073} C_VEL
LIN {X 0,Y 180.188,Z 284.309,A -85,B 0,C 180,E1 -23315.036,E2 -23315.036} C_VEL
LIN {X 0,Y 178.614,Z 296.603,A -85,B 0,C 180,E1 -23316.355,E2 -23316.355} C_VEL
LIN {X 0,Y 176.665,Z 308.225,A -85,B 0,C 180,E1 -23318.033,E2 -23318.033} C_VEL
LIN {X 0,Y 174.235,Z 319.654,A -85,B 0,C 180,E1 -23320.166,E2 -23320.166} C_VEL
LIN {X 0,Y 171.689,Z 330.269,A -85,B 0,C 180,E1 -23322.695,E2 -23322.695} C_VEL
LIN {X 0,Y 169.272,Z 339.984,A -85,B 0,C 180,E1 -23325.658,E2 -23325.658} C_VEL
LIN {X 0,Y 166.944,Z 348.772,A -85,B 0,C 180,E1 -23329.043,E2 -23329.043} C_VEL
LIN {X 0,Y 165.139,Z 355.932,A -85,B 0,C 180,E1 -23332.523,E2 -23332.523} C_VEL
LIN {X 0,Y 163.793,Z 361.174,A -85,B 0,C 180,E1 -23335.705,E2 -23335.705} C_VEL
LIN {X 0,Y 162.766,Z 365.804,A -85,B 0,C 180,E1 -23339.223,E2 -23339.223} C_VEL
LIN {X 0,Y 162.024,Z 369.469,A -85,B 0,C 180,E1 -23342.836,E2 -23342.836} C_VEL
LIN {X 0,Y 161.637,Z 372.791,A -85,B 0,C 180,E1 -23347.499,E2 -23347.499} C_VEL
LIN {X 0,Y 162.044,Z 374.681,A -85,B 0,C 180,E1 -23352.5,E2 -23352.5} C_VEL
LIN {X 0,Y 163.171,Z 375.045,A -85,B 0,C 180,E1 -23357.074,E2 -23357.074} C_VEL
LIN {X 0,Y 164.491,Z 374.463,A -85,B 0,C 180,E1 -23360.272,E2 -23360.272} C_VEL
LIN {X 0,Y 166.336,Z 373.074,A -85,B 0,C 180,E1 -23363.736,E2 -23363.736} C_VEL
LIN {X 0,Y 169.708,Z 369.757,A -85,B 0,C 180,E1 -23368.387,E2 -23368.387} C_VEL
LIN {X 0,Y 172.721,Z 366.354,A -85,B 0,C 180,E1 -23371.56,E2 -23371.56} C_VEL
LIN {X 0,Y 176.208,Z 361.99,A -85,B 0,C 180,E1 -23374.629,E2 -23374.629} C_VEL
LIN {X 0,Y 180.129,Z 356.573,A -85,B 0,C 180,E1 -23377.569,E2 -23377.569} C_VEL
LIN {X 0,Y 184.561,Z 349.91,A -85,B 0,C 180,E1 -23380.362,E2 -23380.362} C_VEL
LIN {X 0,Y 189.811,Z 340.921,A -85,B 0,C 180,E1 -23383.302,E2 -23383.302} C_VEL
LIN {X 0,Y 194.964,Z 330.781,A -85,B 0,C 180,E1 -23385.776,E2 -23385.776} C_VEL
LIN {X 0,Y 199.587,Z 320.041,A -85,B 0,C 180,E1 -23387.804,E2 -23387.804} C_VEL
LIN {X 0,Y 203.372,Z 309.492,A -85,B 0,C 180,E1 -23389.341,E2 -23389.341} C_VEL
LIN {X 0,Y 206.589,Z 298.312,A -85,B 0,C 180,E1 -23390.603,E2 -23390.603} C_VEL
LIN {X 0,Y 209.398,Z 285.464,A -85,B 0,C 180,E1 -23391.68,E2 -23391.68} C_VEL
LIN {X 0,Y 211.343,Z 273.215,A -85,B 0,C 180,E1 -23392.357,E2 -23392.357} C_VEL
LIN {X 0,Y 214.619,Z 237.92,A -85,B 0,C 180,E1 -23393.641,E2 -23393.641} C_VEL
LIN {X 0,Y 211.547,Z 231.659,A -85,B 0,C 180,E1 -23395.52,E2 -23395.52} C_VEL
LIN {X 0,Y 207.381,Z 223.958,A -85,B 0,C 180,E1 -23398.362,E2 -23398.362} C_VEL
LIN {X 0,Y 205.198,Z 220.566,A -85,B 0,C 180,E1 -23400.001,E2 -23400.001} C_VEL
LIN {X 0,Y 202.018,Z 215.274,A -85,B 0,C 180,E1 -23402.824,E2 -23402.824} C_VEL
LIN {X 0,Y 200.62,Z 213.046,A -85,B 0,C 180,E1 -23404.239,E2 -23404.239} C_VEL
LIN {X 0,Y 198.166,Z 209.95,A -85,B 0,C 180,E1 -23407.092,E2 -23407.092} C_VEL
LIN {X 0,Y 197.424,Z 208.583,A -85,B 0,C 180,E1 -23408.188,E2 -23408.188} C_VEL
LIN {X 0,Y 194.434,Z 204.791,A -85,B 0,C 180,E1 -23414.527,E2 -23414.527} C_VEL
LIN {X 0,Y 194.267,Z 204.226,A -85,B 0,C 180,E1 -23415.511,E2 -23415.511} C_VEL
LIN {X 0,Y 193.875,Z 204.489,A -85,B 0,C 180,E1 -23419.52,E2 -23419.52} C_VEL
LIN {X 0,Y 194.799,Z 206.173,A -85,B 0,C 180,E1 -23424.306,E2 -23424.306} C_VEL
LIN {X 0,Y 198.478,Z 212.782,A -85,B 0,C 180,E1 -23431.04,E2 -23431.04} C_VEL
LIN {X 0,Y 201.561,Z 218.661,A -85,B 0,C 180,E1 -23434.557,E2 -23434.557} C_VEL
LIN {X 0,Y 204.465,Z 224.393,A -85,B 0,C 180,E1 -23437.24,E2 -23437.24} C_VEL
LIN {X 0,Y 206.827,Z 229.348,A -85,B 0,C 180,E1 -23439.147,E2 -23439.147} C_VEL
LIN {X 0,Y 209.608,Z 235.563,A -85,B 0,C 180,E1 -23441.172,E2 -23441.172} C_VEL
LIN {X 0,Y 212.364,Z 242.637,A -85,B 0,C 180,E1 -23443.04,E2 -23443.04} C_VEL
LIN {X 0,Y 213.907,Z 247.493,A -85,B 0,C 180,E1 -23444.09,E2 -23444.09} C_VEL
LIN {X 0,Y 211.977,Z 269.46,A -85,B 0,C 180,E1 -23444.879,E2 -23444.879} C_VEL
LIN {X 0,Y 210.09,Z 287.003,A -85,B 0,C 180,E1 -23445.548,E2 -23445.548} C_VEL
LIN {X 0,Y 207.545,Z 300.281,A -85,B 0,C 180,E1 -23446.308,E2 -23446.308} C_VEL
LIN {X 0,Y 203.966,Z 313.665,A -85,B 0,C 180,E1 -23447.45,E2 -23447.45} C_VEL
LIN {X 0,Y 200.059,Z 325.209,A -85,B 0,C 180,E1 -23448.799,E2 -23448.799} C_VEL
LIN {X 0,Y 195.171,Z 336.877,A -85,B 0,C 180,E1 -23450.603,E2 -23450.603} C_VEL
LIN {X 0,Y 190.626,Z 346.343,A -85,B 0,C 180,E1 -23452.53,E2 -23452.53} C_VEL
LIN {X 0,Y 188.25,Z 350.791,A -85,B 0,C 180,E1 -23453.607,E2 -23453.607} C_VEL
LIN {X 0,Y 185.452,Z 354.921,A -85,B 0,C 180,E1 -23454.587,E2 -23454.587} C_VEL
LIN {X 0,Y 179.478,Z 361.332,A -85,B 0,C 180,E1 -23456.054,E2 -23456.054} C_VEL
LIN {X 0,Y 173.455,Z 367.103,A -85,B 0,C 180,E1 -23457.776,E2 -23457.776} C_VEL
LIN {X 0,Y 170.641,Z 370.225,A -85,B 0,C 180,E1 -23459.151,E2 -23459.151} C_VEL
LIN {X 0,Y 165.649,Z 376.911,A -85,B 0,C 180,E1 -23463.199,E2 -23463.199} C_VEL
LIN {X 0,Y 161.828,Z 381.501,A -85,B 0,C 180,E1 -23466.99,E2 -23466.99} C_VEL
LIN {X 0,Y 159.942,Z 383.726,A -85,B 0,C 180,E1 -23469.418,E2 -23469.418} C_VEL
LIN {X 0,Y 156.89,Z 386.895,A -85,B 0,C 180,E1 -23474.407,E2 -23474.407} C_VEL
LIN {X 0,Y 155.311,Z 388.539,A -85,B 0,C 180,E1 -23479.57,E2 -23479.57} C_VEL
LIN {X 0,Y 154.839,Z 388.59,A -85,B 0,C 180,E1 -23484.79,E2 -23484.79} C_VEL
LIN {X 0,Y 154.914,Z 388.04,A -85,B 0,C 180,E1 -23487.398,E2 -23487.398} C_VEL
LIN {X 0,Y 155.189,Z 387.1,A -85,B 0,C 180,E1 -23489.998,E2 -23489.998} C_VEL
LIN {X 0,Y 154.949,Z 384.883,A -85,B 0,C 180,E1 -23493.738,E2 -23493.738} C_VEL
LIN {X 0,Y 155.115,Z 381.407,A -85,B 0,C 180,E1 -23497.811,E2 -23497.811} C_VEL
LIN {X 0,Y 155.643,Z 376.892,A -85,B 0,C 180,E1 -23501.722,E2 -23501.722} C_VEL
LIN {X 0,Y 157.057,Z 369.986,A -85,B 0,C 180,E1 -23506.239,E2 -23506.239} C_VEL
LIN {X 0,Y 158.954,Z 362.44,A -85,B 0,C 180,E1 -23510.037,E2 -23510.037} C_VEL
LIN {X 0,Y 161.199,Z 353.831,A -85,B 0,C 180,E1 -23513.458,E2 -23513.458} C_VEL
LIN {X 0,Y 163.795,Z 344.258,A -85,B 0,C 180,E1 -23516.432,E2 -23516.432} C_VEL
LIN {X 0,Y 166.202,Z 334.913,A -85,B 0,C 180,E1 -23518.749,E2 -23518.749} C_VEL
LIN {X 0,Y 168.889,Z 323.402,A -85,B 0,C 180,E1 -23520.993,E2 -23520.993} C_VEL
LIN {X 0,Y 171.259,Z 311.38,A -85,B 0,C 180,E1 -23522.762,E2 -23522.762} C_VEL
LIN {X 0,Y 173.105,Z 299.746,A -85,B 0,C 180,E1 -23524.021,E2 -23524.021} C_VEL
LIN {X 0,Y 174.706,Z 286.242,A -85,B 0,C 180,E1 -23525.016,E2 -23525.016} C_VEL
LIN {X 0,Y 177.332,Z 240.643,A -85,B 0,C 180,E1 -23527.041,E2 -23527.041} C_VEL
LIN {X 0,Y 175.067,Z 218.592,A -85,B 0,C 180,E1 -23528.594,E2 -23528.594} C_VEL
LIN {X 0,Y 167.987,Z 199.157,A -85,B 0,C 180,E1 -23531.028,E2 -23531.028} C_VEL
LIN {X 0,Y 161.488,Z 184.273,A -85,B 0,C 180,E1 -23533.312,E2 -23533.312} C_VEL
LIN {X 0,Y 157.864,Z 176.419,A -85,B 0,C 180,E1 -23534.671,E2 -23534.671} C_VEL
LIN {X 0,Y 157.245,Z 173.898,A -85,B 0,C 180,E1 -23536.385,E2 -23536.385} C_VEL
LIN {X 0,Y 157.206,Z 173.901,A -85,B 0,C 180,E1 -23541.251,E2 -23541.251} C_VEL
LIN {X 0,Y 157.278,Z 173.895,A -85,B 0,C 180,E1 -23544.484,E2 -23544.484} C_VEL
LIN {X 0,Y 157.301,Z 173.893,A -85,B 0,C 180,E1 -23548.089,E2 -23548.089} C_VEL
LIN {X 0,Y 157.322,Z 173.889,A -85,B 0,C 180,E1 -23553.465,E2 -23553.465} C_VEL
LIN {X 0,Y 157.377,Z 173.882,A -85,B 0,C 180,E1 -23559.682,E2 -23559.682} C_VEL
LIN {X 0,Y 157.422,Z 173.866,A -85,B 0,C 180,E1 -23564.461,E2 -23564.461} C_VEL
LIN {X 0,Y 157.724,Z 173.834,A -85,B 0,C 180,E1 -23569.732,E2 -23569.732} C_VEL
LIN {X 0,Y 157.806,Z 173.811,A -85,B 0,C 180,E1 -23572.321,E2 -23572.321} C_VEL
LIN {X 0,Y 158.257,Z 173.764,A -85,B 0,C 180,E1 -23579.999,E2 -23579.999} C_VEL
LIN {X 0,Y 157.806,Z 173.827,A -85,B 0,C 180,E1 -23587.677,E2 -23587.677} C_VEL
LIN {X 0,Y 157.68,Z 173.834,A -85,B 0,C 180,E1 -23591.321,E2 -23591.321} C_VEL
LIN {X 0,Y 157.476,Z 173.854,A -85,B 0,C 180,E1 -23595.53,E2 -23595.53} C_VEL
LIN {X 0,Y 157.367,Z 173.879,A -85,B 0,C 180,E1 -23600.932,E2 -23600.932} C_VEL
LIN {X 0,Y 157.311,Z 173.867,A -85,B 0,C 180,E1 -23606.684,E2 -23606.684} C_VEL
LIN {X 0,Y 157.274,Z 173.887,A -85,B 0,C 180,E1 -23612.426,E2 -23612.426} C_VEL
LIN {X 0,Y 157.322,Z 173.866,A -85,B 0,C 180,E1 -23616.478,E2 -23616.478} C_VEL
LIN {X 0,Y 157.294,Z 173.888,A -85,B 0,C 180,E1 -23622.081,E2 -23622.081} C_VEL
LIN {X 0,Y 157.311,Z 173.873,A -85,B 0,C 180,E1 -23625.626,E2 -23625.626} C_VEL
LIN {X 0,Y 157.29,Z 173.891,A -85,B 0,C 180,E1 -23631.28,E2 -23631.28} C_VEL
LIN {X 0,Y 157.291,Z 173.879,A -85,B 0,C 180,E1 -23634.491,E2 -23634.491} C_VEL
LIN {X 0,Y 157.298,Z 173.892,A -85,B 0,C 180,E1 -23638.091,E2 -23638.091} C_VEL
LIN {X 0,Y 157.318,Z 173.888,A -85,B 0,C 180,E1 -23643.467,E2 -23643.467} C_VEL
LIN {X 0,Y 157.39,Z 173.88,A -85,B 0,C 180,E1 -23649.668,E2 -23649.668} C_VEL
LIN {X 0,Y 157.474,Z 173.872,A -85,B 0,C 180,E1 -23654.469,E2 -23654.469} C_VEL
LIN {X 0,Y 157.769,Z 173.836,A -85,B 0,C 180,E1 -23659.737,E2 -23659.737} C_VEL
LIN {X 0,Y 157.73,Z 173.841,A -85,B 0,C 180,E1 -23664.007,E2 -23664.007} C_VEL
LIN {X 0,Y 158.767,Z 176.707,A -85,B 0,C 180,E1 -23664.449,E2 -23664.449} C_VEL
LIN {X 0,Y 165.924,Z 188.674,A -85,B 0,C 180,E1 -23666.773,E2 -23666.773} C_VEL
LIN {X 0,Y 176.442,Z 211.795,A -85,B 0,C 180,E1 -23670.132,E2 -23670.132} C_VEL
LIN {X 0,Y 178.451,Z 216.967,A -85,B 0,C 180,E1 -23670.756,E2 -23670.756} C_VEL
LIN {X 0,Y 175.117,Z 271.238,A -85,B 0,C 180,E1 -23673.103,E2 -23673.103} C_VEL
LIN {X 0,Y 173.704,Z 284.63,A -85,B 0,C 180,E1 -23674.102,E2 -23674.102} C_VEL
LIN {X 0,Y 171.94,Z 297.762,A -85,B 0,C 180,E1 -23675.572,E2 -23675.572} C_VEL
LIN {X 0,Y 169.819,Z 309.691,A -85,B 0,C 180,E1 -23677.402,E2 -23677.402} C_VEL
LIN {X 0,Y 167.208,Z 321.232,A -85,B 0,C 180,E1 -23679.68,E2 -23679.68} C_VEL
LIN {X 0,Y 164.621,Z 331.633,A -85,B 0,C 180,E1 -23682.327,E2 -23682.327} C_VEL
LIN {X 0,Y 162.003,Z 341.607,A -85,B 0,C 180,E1 -23685.579,E2 -23685.579} C_VEL
LIN {X 0,Y 159.579,Z 350.548,A -85,B 0,C 180,E1 -23689.289,E2 -23689.289} C_VEL
LIN {X 0,Y 157.691,Z 357.621,A -85,B 0,C 180,E1 -23693.061,E2 -23693.061} C_VEL
LIN {X 0,Y 156.363,Z 363.044,A -85,B 0,C 180,E1 -23696.711,E2 -23696.711} C_VEL
LIN {X 0,Y 155.321,Z 367.674,A -85,B 0,C 180,E1 -23700.718,E2 -23700.718} C_VEL
LIN {X 0,Y 154.608,Z 371.387,A -85,B 0,C 180,E1 -23705.095,E2 -23705.095} C_VEL
LIN {X 0,Y 154.616,Z 373.88,A -85,B 0,C 180,E1 -23709.523,E2 -23709.523} C_VEL
LIN {X 0,Y 155.119,Z 375.11,A -85,B 0,C 180,E1 -23713.541,E2 -23713.541} C_VEL
LIN {X 0,Y 156.198,Z 375.401,A -85,B 0,C 180,E1 -23717.555,E2 -23717.555} C_VEL
LIN {X 0,Y 157.872,Z 374.766,A -85,B 0,C 180,E1 -23721.449,E2 -23721.449} C_VEL
LIN {X 0,Y 160.704,Z 372.707,A -85,B 0,C 180,E1 -23726.196,E2 -23726.196} C_VEL
LIN {X 0,Y 164.577,Z 369.02,A -85,B 0,C 180,E1 -23730.839,E2 -23730.839} C_VEL
LIN {X 0,Y 168.873,Z 364.28,A -85,B 0,C 180,E1 -23734.805,E2 -23734.805} C_VEL
LIN {X 0,Y 173.758,Z 358.204,A -85,B 0,C 180,E1 -23738.483,E2 -23738.483} C_VEL
LIN {X 0,Y 178.944,Z 350.957,A -85,B 0,C 180,E1 -23741.689,E2 -23741.689} C_VEL
LIN {X 0,Y 184.085,Z 342.695,A -85,B 0,C 180,E1 -23744.501,E2 -23744.501} C_VEL
LIN {X 0,Y 189.326,Z 333.252,A -85,B 0,C 180,E1 -23746.935,E2 -23746.935} C_VEL
LIN {X 0,Y 194.32,Z 322.465,A -85,B 0,C 180,E1 -23749.068,E2 -23749.068} C_VEL
LIN {X 0,Y 198.67,Z 311.25,A -85,B 0,C 180,E1 -23750.785,E2 -23750.785} C_VEL
LIN {X 0,Y 202.28,Z 299.67,A -85,B 0,C 180,E1 -23752.14,E2 -23752.14} C_VEL
LIN {X 0,Y 205.255,Z 287.124,A -85,B 0,C 180,E1 -23753.211,E2 -23753.211} C_VEL
LIN {X 0,Y 207.297,Z 275.13,A -85,B 0,C 180,E1 -23753.92,E2 -23753.92} C_VEL
LIN {X 0,Y 210.659,Z 241.191,A -85,B 0,C 180,E1 -23755.173,E2 -23755.173} C_VEL
LIN {X 0,Y 206.608,Z 232.978,A -85,B 0,C 180,E1 -23757.956,E2 -23757.956} C_VEL
LIN {X 0,Y 203.568,Z 227.561,A -85,B 0,C 180,E1 -23760.315,E2 -23760.315} C_VEL
LIN {X 0,Y 199.944,Z 221.363,A -85,B 0,C 180,E1 -23763.712,E2 -23763.712} C_VEL
LIN {X 0,Y 199.009,Z 219.763,A -85,B 0,C 180,E1 -23764.719,E2 -23764.719} C_VEL
LIN {X 0,Y 196.552,Z 216.409,A -85,B 0,C 180,E1 -23767.809,E2 -23767.809} C_VEL
LIN {X 0,Y 195.937,Z 215.364,A -85,B 0,C 180,E1 -23768.756,E2 -23768.756} C_VEL
LIN {X 0,Y 193.21,Z 211.251,A -85,B 0,C 180,E1 -23775.598,E2 -23775.598} C_VEL
LIN {X 0,Y 192.868,Z 211.631,A -85,B 0,C 180,E1 -23779.99,E2 -23779.99} C_VEL
LIN {X 0,Y 193.679,Z 213.156,A -85,B 0,C 180,E1 -23784.112,E2 -23784.112} C_VEL
LIN {X 0,Y 196.927,Z 219.449,A -85,B 0,C 180,E1 -23790.466,E2 -23790.466} C_VEL
LIN {X 0,Y 199.602,Z 224.955,A -85,B 0,C 180,E1 -23793.783,E2 -23793.783} C_VEL
LIN {X 0,Y 202.247,Z 230.551,A -85,B 0,C 180,E1 -23796.447,E2 -23796.447} C_VEL
LIN {X 0,Y 204.734,Z 235.995,A -85,B 0,C 180,E1 -23798.559,E2 -23798.559} C_VEL
LIN {X 0,Y 208.007,Z 244.177,A -85,B 0,C 180,E1 -23801.098,E2 -23801.098} C_VEL
LIN {X 0,Y 209.971,Z 250.071,A -85,B 0,C 180,E1 -23802.523,E2 -23802.523} C_VEL
LIN {X 0,Y 209.154,Z 259.916,A -85,B 0,C 180,E1 -23802.924,E2 -23802.924} C_VEL
LIN {X 0,Y 206.477,Z 285.136,A -85,B 0,C 180,E1 -23803.83,E2 -23803.83} C_VEL
LIN {X 0,Y 203.986,Z 298.252,A -85,B 0,C 180,E1 -23804.539,E2 -23804.539} C_VEL
LIN {X 0,Y 200.649,Z 310.736,A -85,B 0,C 180,E1 -23805.529,E2 -23805.529} C_VEL
LIN {X 0,Y 196.579,Z 322.722,A -85,B 0,C 180,E1 -23806.861,E2 -23806.861} C_VEL
LIN {X 0,Y 192.039,Z 333.683,A -85,B 0,C 180,E1 -23808.445,E2 -23808.445} C_VEL
LIN {X 0,Y 187.152,Z 343.696,A -85,B 0,C 180,E1 -23810.326,E2 -23810.326} C_VEL
LIN {X 0,Y 182.071,Z 352.79,A -85,B 0,C 180,E1 -23812.557,E2 -23812.557} C_VEL
LIN {X 0,Y 176.58,Z 361.699,A -85,B 0,C 180,E1 -23815.446,E2 -23815.446} C_VEL
LIN {X 0,Y 171.579,Z 368.953,A -85,B 0,C 180,E1 -23818.515,E2 -23818.515} C_VEL
LIN {X 0,Y 170.641,Z 370.225,A -85,B 0,C 180,E1 -23819.151,E2 -23819.151} C_VEL
LIN {X 0,Y 167.858,Z 373.178,A -85,B 0,C 180,E1 -23820.629,E2 -23820.629} C_VEL
LIN {X 0,Y 161.962,Z 377.538,A -85,B 0,C 180,E1 -23822.964,E2 -23822.964} C_VEL
LIN {X 0,Y 156.34,Z 381.138,A -85,B 0,C 180,E1 -23825.584,E2 -23825.584} C_VEL
LIN {X 0,Y 154.058,Z 382.922,A -85,B 0,C 180,E1 -23827.475,E2 -23827.475} C_VEL
LIN {X 0,Y 151.502,Z 385.444,A -85,B 0,C 180,E1 -23831.05,E2 -23831.05} C_VEL
LIN {X 0,Y 150.028,Z 386.774,A -85,B 0,C 180,E1 -23833.674,E2 -23833.674} C_VEL
LIN {X 0,Y 149.022,Z 387.715,A -85,B 0,C 180,E1 -23836.359,E2 -23836.359} C_VEL
LIN {X 0,Y 147.879,Z 388.395,A -85,B 0,C 180,E1 -23841.801,E2 -23841.801} C_VEL
LIN {X 0,Y 147.847,Z 387.576,A -85,B 0,C 180,E1 -23847.274,E2 -23847.274} C_VEL
LIN {X 0,Y 148.102,Z 386.547,A -85,B 0,C 180,E1 -23849.998,E2 -23849.998} C_VEL
LIN {X 0,Y 147.885,Z 384.449,A -85,B 0,C 180,E1 -23853.609,E2 -23853.609} C_VEL
LIN {X 0,Y 148.052,Z 380.636,A -85,B 0,C 180,E1 -23858.186,E2 -23858.186} C_VEL
LIN {X 0,Y 148.647,Z 375.975,A -85,B 0,C 180,E1 -23862.283,E2 -23862.283} C_VEL
LIN {X 0,Y 150.241,Z 368.888,A -85,B 0,C 180,E1 -23866.998,E2 -23866.998} C_VEL
LIN {X 0,Y 152.263,Z 361.166,A -85,B 0,C 180,E1 -23870.958,E2 -23870.958} C_VEL
LIN {X 0,Y 154.41,Z 353.217,A -85,B 0,C 180,E1 -23874.18,E2 -23874.18} C_VEL
LIN {X 0,Y 157.129,Z 343.528,A -85,B 0,C 180,E1 -23877.286,E2 -23877.286} C_VEL
LIN {X 0,Y 159.623,Z 334.094,A -85,B 0,C 180,E1 -23879.689,E2 -23879.689} C_VEL
LIN {X 0,Y 162.465,Z 322.491,A -85,B 0,C 180,E1 -23881.998,E2 -23881.998} C_VEL
LIN {X 0,Y 164.917,Z 310.227,A -85,B 0,C 180,E1 -23883.824,E2 -23883.824} C_VEL
LIN {X 0,Y 167.016,Z 296.855,A -85,B 0,C 180,E1 -23885.258,E2 -23885.258} C_VEL
LIN {X 0,Y 168.456,Z 284.041,A -85,B 0,C 180,E1 -23886.154,E2 -23886.154} C_VEL
LIN {X 0,Y 170.99,Z 241.241,A -85,B 0,C 180,E1 -23888.094,E2 -23888.094} C_VEL
LIN {X 0,Y 169.058,Z 221.085,A -85,B 0,C 180,E1 -23889.567,E2 -23889.567} C_VEL
LIN {X 0,Y 162.511,Z 202.821,A -85,B 0,C 180,E1 -23891.971,E2 -23891.971} C_VEL
LIN {X 0,Y 156.184,Z 188.117,A -85,B 0,C 180,E1 -23894.304,E2 -23894.304} C_VEL
LIN {X 0,Y 151.776,Z 179.065,A -85,B 0,C 180,E1 -23896.005,E2 -23896.005} C_VEL
LIN {X 0,Y 150.479,Z 176.043,A -85,B 0,C 180,E1 -23896.579,E2 -23896.579} C_VEL
LIN {X 0,Y 150.165,Z 174.78,A -85,B 0,C 180,E1 -23897.503,E2 -23897.503} C_VEL
LIN {X 0,Y 150.179,Z 174.781,A -85,B 0,C 180,E1 -23902.706,E2 -23902.706} C_VEL
LIN {X 0,Y 150.22,Z 174.776,A -85,B 0,C 180,E1 -23907.363,E2 -23907.363} C_VEL
LIN {X 0,Y 150.245,Z 174.769,A -85,B 0,C 180,E1 -23912.715,E2 -23912.715} C_VEL
LIN {X 0,Y 150.339,Z 174.759,A -85,B 0,C 180,E1 -23919.217,E2 -23919.217} C_VEL
LIN {X 0,Y 150.329,Z 174.747,A -85,B 0,C 180,E1 -23923.708,E2 -23923.708} C_VEL
LIN {X 0,Y 150.645,Z 174.717,A -85,B 0,C 180,E1 -23929.243,E2 -23929.243} C_VEL
LIN {X 0,Y 150.74,Z 174.691,A -85,B 0,C 180,E1 -23931.958,E2 -23931.958} C_VEL
LIN {X 0,Y 151.217,Z 174.64,A -85,B 0,C 180,E1 -23939.999,E2 -23939.999} C_VEL
LIN {X 0,Y 150.742,Z 174.707,A -85,B 0,C 180,E1 -23948.039,E2 -23948.039} C_VEL
LIN {X 0,Y 150.611,Z 174.713,A -85,B 0,C 180,E1 -23951.506,E2 -23951.506} C_VEL
LIN {X 0,Y 150.38,Z 174.741,A -85,B 0,C 180,E1 -23956.283,E2 -23956.283} C_VEL
LIN {X 0,Y 150.348,Z 174.753,A -85,B 0,C 180,E1 -23960.793,E2 -23960.793} C_VEL
LIN {X 0,Y 150.24,Z 174.752,A -85,B 0,C 180,E1 -23967.282,E2 -23967.282} C_VEL
LIN {X 0,Y 150.215,Z 174.765,A -85,B 0,C 180,E1 -23972.634,E2 -23972.634} C_VEL
LIN {X 0,Y 150.234,Z 174.751,A -85,B 0,C 180,E1 -23977.454,E2 -23977.454} C_VEL
LIN {X 0,Y 150.236,Z 174.767,A -85,B 0,C 180,E1 -23981.544,E2 -23981.544} C_VEL
LIN {X 0,Y 150.286,Z 174.748,A -85,B 0,C 180,E1 -23985.458,E2 -23985.458} C_VEL
LIN {X 0,Y 150.237,Z 174.767,A -85,B 0,C 180,E1 -23989.089,E2 -23989.089} C_VEL
LIN {X 0,Y 150.237,Z 174.766,A -85,B 0,C 180,E1 -23992.676,E2 -23992.676} C_VEL
LIN {X 0,Y 150.219,Z 174.771,A -85,B 0,C 180,E1 -23997.363,E2 -23997.363} C_VEL
LIN {X 0,Y 150.241,Z 174.77,A -85,B 0,C 180,E1 -24002.718,E2 -24002.718} C_VEL
LIN {X 0,Y 150.347,Z 174.758,A -85,B 0,C 180,E1 -24009.208,E2 -24009.208} C_VEL
LIN {X 0,Y 150.379,Z 174.757,A -85,B 0,C 180,E1 -24013.717,E2 -24013.717} C_VEL
LIN {X 0,Y 150.685,Z 174.72,A -85,B 0,C 180,E1 -24019.249,E2 -24019.249} C_VEL
LIN {X 0,Y 150.78,Z 174.706,A -85,B 0,C 180,E1 -24022.227,E2 -24022.227} C_VEL
LIN {X 0,Y 151.837,Z 177.71,A -85,B 0,C 180,E1 -24022.766,E2 -24022.766} C_VEL
LIN {X 0,Y 153.213,Z 179.985,A -85,B 0,C 180,E1 -24023.279,E2 -24023.279} C_VEL
LIN {X 0,Y 161.093,Z 193.605,A -85,B 0,C 180,E1 -24026.027,E2 -24026.027} C_VEL
LIN {X 0,Y 170.789,Z 215.259,A -85,B 0,C 180,E1 -24029.278,E2 -24029.278} C_VEL
LIN {X 0,Y 172.14,Z 218.831,A -85,B 0,C 180,E1 -24029.73,E2 -24029.73} C_VEL
LIN {X 0,Y 168.737,Z 271.558,A -85,B 0,C 180,E1 -24032.075,E2 -24032.075} C_VEL
LIN {X 0,Y 167.31,Z 284.741,A -85,B 0,C 180,E1 -24033.087,E2 -24033.087} C_VEL
LIN {X 0,Y 165.498,Z 297.687,A -85,B 0,C 180,E1 -24034.568,E2 -24034.568} C_VEL
LIN {X 0,Y 163.245,Z 309.902,A -85,B 0,C 180,E1 -24036.492,E2 -24036.492} C_VEL
LIN {X 0,Y 160.564,Z 321.309,A -85,B 0,C 180,E1 -24038.814,E2 -24038.814} C_VEL
LIN {X 0,Y 157.845,Z 331.948,A -85,B 0,C 180,E1 -24041.616,E2 -24041.616} C_VEL
LIN {X 0,Y 155.012,Z 342.234,A -85,B 0,C 180,E1 -24045.113,E2 -24045.113} C_VEL
LIN {X 0,Y 152.611,Z 350.756,A -85,B 0,C 180,E1 -24048.807,E2 -24048.807} C_VEL
LIN {X 0,Y 150.687,Z 357.675,A -85,B 0,C 180,E1 -24052.632,E2 -24052.632} C_VEL
LIN {X 0,Y 149.282,Z 363.29,A -85,B 0,C 180,E1 -24056.56,E2 -24056.56} C_VEL
LIN {X 0,Y 148.054,Z 368.621,A -85,B 0,C 180,E1 -24061.479,E2 -24061.479} C_VEL
LIN {X 0,Y 147.47,Z 372.035,A -85,B 0,C 180,E1 -24065.89,E2 -24065.89} C_VEL
LIN {X 0,Y 147.564,Z 374.338,A -85,B 0,C 180,E1 -24070.359,E2 -24070.359} C_VEL
LIN {X 0,Y 148.394,Z 375.613,A -85,B 0,C 180,E1 -24075.27,E2 -24075.27} C_VEL
LIN {X 0,Y 149.551,Z 375.738,A -85,B 0,C 180,E1 -24078.861,E2 -24078.861} C_VEL
LIN {X 0,Y 151.423,Z 375.027,A -85,B 0,C 180,E1 -24082.89,E2 -24082.89} C_VEL
LIN {X 0,Y 153.807,Z 373.448,A -85,B 0,C 180,E1 -24086.75,E2 -24086.75} C_VEL
LIN {X 0,Y 156.804,Z 370.991,A -85,B 0,C 180,E1 -24090.462,E2 -24090.462} C_VEL
LIN {X 0,Y 160.408,Z 367.589,A -85,B 0,C 180,E1 -24094.017,E2 -24094.017} C_VEL
LIN {X 0,Y 164.525,Z 363.177,A -85,B 0,C 180,E1 -24097.392,E2 -24097.392} C_VEL
LIN {X 0,Y 169.165,Z 357.617,A -85,B 0,C 180,E1 -24100.589,E2 -24100.589} C_VEL
LIN {X 0,Y 174.37,Z 350.664,A -85,B 0,C 180,E1 -24103.614,E2 -24103.614} C_VEL
LIN {X 0,Y 179.85,Z 342.262,A -85,B 0,C 180,E1 -24106.441,E2 -24106.441} C_VEL
LIN {X 0,Y 185.418,Z 332.566,A -85,B 0,C 180,E1 -24108.884,E2 -24108.884} C_VEL
LIN {X 0,Y 190.401,Z 322.227,A -85,B 0,C 180,E1 -24110.897,E2 -24110.897} C_VEL
LIN {X 0,Y 195.016,Z 310.676,A -85,B 0,C 180,E1 -24112.633,E2 -24112.633} C_VEL
LIN {X 0,Y 198.781,Z 298.717,A -85,B 0,C 180,E1 -24113.979,E2 -24113.979} C_VEL
LIN {X 0,Y 201.881,Z 285.704,A -85,B 0,C 180,E1 -24115.048,E2 -24115.048} C_VEL
LIN {X 0,Y 204.01,Z 273.039,A -85,B 0,C 180,E1 -24115.717,E2 -24115.717} C_VEL
LIN {X 0,Y 206.847,Z 244.609,A -85,B 0,C 180,E1 -24116.768,E2 -24116.768} C_VEL
LIN {X 0,Y 202.898,Z 236.372,A -85,B 0,C 180,E1 -24119.833,E2 -24119.833} C_VEL
LIN {X 0,Y 200.306,Z 231.947,A -85,B 0,C 180,E1 -24122.108,E2 -24122.108} C_VEL
LIN {X 0,Y 197.953,Z 227.479,A -85,B 0,C 180,E1 -24124.585,E2 -24124.585} C_VEL
LIN {X 0,Y 197.093,Z 226.133,A -85,B 0,C 180,E1 -24125.593,E2 -24125.593} C_VEL
LIN {X 0,Y 194.88,Z 222.672,A -85,B 0,C 180,E1 -24128.676,E2 -24128.676} C_VEL
LIN {X 0,Y 192.145,Z 218.284,A -85,B 0,C 180,E1 -24135.686,E2 -24135.686} C_VEL
LIN {X 0,Y 191.805,Z 218.588,A -85,B 0,C 180,E1 -24139.68,E2 -24139.68} C_VEL
LIN {X 0,Y 192.526,Z 220.109,A -85,B 0,C 180,E1 -24143.838,E2 -24143.838} C_VEL
LIN {X 0,Y 195.386,Z 226.122,A -85,B 0,C 180,E1 -24149.884,E2 -24149.884} C_VEL
LIN {X 0,Y 197.737,Z 231.374,A -85,B 0,C 180,E1 -24153.061,E2 -24153.061} C_VEL
LIN {X 0,Y 200.295,Z 237.104,A -85,B 0,C 180,E1 -24155.81,E2 -24155.81} C_VEL
LIN {X 0,Y 202.88,Z 243.326,A -85,B 0,C 180,E1 -24158.162,E2 -24158.162} C_VEL
LIN {X 0,Y 205.781,Z 251.507,A -85,B 0,C 180,E1 -24160.596,E2 -24160.596} C_VEL
LIN {X 0,Y 206.273,Z 253.24,A -85,B 0,C 180,E1 -24160.994,E2 -24160.994} C_VEL
LIN {X 0,Y 202.926,Z 284.296,A -85,B 0,C 180,E1 -24162.082,E2 -24162.082} C_VEL
LIN {X 0,Y 200.461,Z 297.199,A -85,B 0,C 180,E1 -24162.771,E2 -24162.771} C_VEL
LIN {X 0,Y 197.022,Z 309.902,A -85,B 0,C 180,E1 -24163.75,E2 -24163.75} C_VEL
LIN {X 0,Y 192.758,Z 321.999,A -85,B 0,C 180,E1 -24165.054,E2 -24165.054} C_VEL
LIN {X 0,Y 188.022,Z 332.975,A -85,B 0,C 180,E1 -24166.618,E2 -24166.618} C_VEL
LIN {X 0,Y 182.907,Z 343.016,A -85,B 0,C 180,E1 -24168.484,E2 -24168.484} C_VEL
LIN {X 0,Y 176.54,Z 353.751,A -85,B 0,C 180,E1 -24171.169,E2 -24171.169} C_VEL
LIN {X 0,Y 170.824,Z 362.45,A -85,B 0,C 180,E1 -24174.105,E2 -24174.105} C_VEL
LIN {X 0,Y 165.6,Z 369.485,A -85,B 0,C 180,E1 -24177.239,E2 -24177.239} C_VEL
LIN {X 0,Y 161.729,Z 374.311,A -85,B 0,C 180,E1 -24180.016,E2 -24180.016} C_VEL
LIN {X 0,Y 157.736,Z 379.034,A -85,B 0,C 180,E1 -24183.54,E2 -24183.54} C_VEL
LIN {X 0,Y 154.058,Z 382.922,A -85,B 0,C 180,E1 -24187.475,E2 -24187.475} C_VEL
LIN {X 0,Y 151.911,Z 384.505,A -85,B 0,C 180,E1 -24189.456,E2 -24189.456} C_VEL
LIN {X 0,Y 147.026,Z 386.437,A -85,B 0,C 180,E1 -24192.681,E2 -24192.681} C_VEL
LIN {X 0,Y 142.638,Z 387.604,A -85,B 0,C 180,E1 -24196.161,E2 -24196.161} C_VEL
LIN {X 0,Y 141.333,Z 387.934,A -85,B 0,C 180,E1 -24198.473,E2 -24198.473} C_VEL
LIN {X 0,Y 140.679,Z 387.756,A -85,B 0,C 180,E1 -24204.264,E2 -24204.264} C_VEL
LIN {X 0,Y 140.739,Z 387.063,A -85,B 0,C 180,E1 -24207.136,E2 -24207.136} C_VEL
LIN {X 0,Y 141.018,Z 385.952,A -85,B 0,C 180,E1 -24209.998,E2 -24209.998} C_VEL
LIN {X 0,Y 140.827,Z 383.977,A -85,B 0,C 180,E1 -24213.503,E2 -24213.503} C_VEL
LIN {X 0,Y 141.01,Z 379.803,A -85,B 0,C 180,E1 -24218.598,E2 -24218.598} C_VEL
LIN {X 0,Y 141.675,Z 375.007,A -85,B 0,C 180,E1 -24222.897,E2 -24222.897} C_VEL
LIN {X 0,Y 143.095,Z 368.91,A -85,B 0,C 180,E1 -24227.137,E2 -24227.137} C_VEL
LIN {X 0,Y 145.198,Z 361.28,A -85,B 0,C 180,E1 -24231.284,E2 -24231.284} C_VEL
LIN {X 0,Y 147.384,Z 353.437,A -85,B 0,C 180,E1 -24234.659,E2 -24234.659} C_VEL
LIN {X 0,Y 150.222,Z 343.884,A -85,B 0,C 180,E1 -24237.893,E2 -24237.893} C_VEL
LIN {X 0,Y 152.792,Z 334.585,A -85,B 0,C 180,E1 -24240.394,E2 -24240.394} C_VEL
LIN {X 0,Y 155.679,Z 323.143,A -85,B 0,C 180,E1 -24242.8,E2 -24242.8} C_VEL
LIN {X 0,Y 158.208,Z 311.27,A -85,B 0,C 180,E1 -24244.69,E2 -24244.69} C_VEL
LIN {X 0,Y 160.281,Z 299.077,A -85,B 0,C 180,E1 -24246.099,E2 -24246.099} C_VEL
LIN {X 0,Y 162.036,Z 285.008,A -85,B 0,C 180,E1 -24247.192,E2 -24247.192} C_VEL
LIN {X 0,Y 164.716,Z 241.808,A -85,B 0,C 180,E1 -24249.227,E2 -24249.227} C_VEL
LIN {X 0,Y 162.849,Z 222.737,A -85,B 0,C 180,E1 -24250.715,E2 -24250.715} C_VEL
LIN {X 0,Y 156.472,Z 205.005,A -85,B 0,C 180,E1 -24253.168,E2 -24253.168} C_VEL
LIN {X 0,Y 151.035,Z 192.153,A -85,B 0,C 180,E1 -24255.326,E2 -24255.326} C_VEL
LIN {X 0,Y 146.558,Z 182.883,A -85,B 0,C 180,E1 -24257.16,E2 -24257.16} C_VEL
LIN {X 0,Y 144.846,Z 179.454,A -85,B 0,C 180,E1 -24257.886,E2 -24257.886} C_VEL
LIN {X 0,Y 143.351,Z 176.868,A -85,B 0,C 180,E1 -24258.509,E2 -24258.509} C_VEL
LIN {X 0,Y 143.102,Z 175.657,A -85,B 0,C 180,E1 -24258.756,E2 -24258.756} C_VEL
LIN {X 0,Y 143.087,Z 175.664,A -85,B 0,C 180,E1 -24263.884,E2 -24263.884} C_VEL
LIN {X 0,Y 143.186,Z 175.652,A -85,B 0,C 180,E1 -24267.321,E2 -24267.321} C_VEL
LIN {X 0,Y 143.191,Z 175.647,A -85,B 0,C 180,E1 -24272.059,E2 -24272.059} C_VEL
LIN {X 0,Y 143.267,Z 175.638,A -85,B 0,C 180,E1 -24278.752,E2 -24278.752} C_VEL
LIN {X 0,Y 143.268,Z 175.627,A -85,B 0,C 180,E1 -24282.881,E2 -24282.881} C_VEL
LIN {X 0,Y 143.592,Z 175.598,A -85,B 0,C 180,E1 -24288.708,E2 -24288.708} C_VEL
LIN {X 0,Y 143.659,Z 175.574,A -85,B 0,C 180,E1 -24291.559,E2 -24291.559} C_VEL
LIN {X 0,Y 144.176,Z 175.516,A -85,B 0,C 180,E1 -24299.998,E2 -24299.998} C_VEL
LIN {X 0,Y 143.662,Z 175.59,A -85,B 0,C 180,E1 -24308.438,E2 -24308.438} C_VEL
LIN {X 0,Y 143.544,Z 175.59,A -85,B 0,C 180,E1 -24311.711,E2 -24311.711} C_VEL
LIN {X 0,Y 143.314,Z 175.626,A -85,B 0,C 180,E1 -24317.11,E2 -24317.11} C_VEL
LIN {X 0,Y 143.274,Z 175.633,A -85,B 0,C 180,E1 -24321.255,E2 -24321.255} C_VEL
LIN {X 0,Y 143.186,Z 175.634,A -85,B 0,C 180,E1 -24327.937,E2 -24327.937} C_VEL
LIN {X 0,Y 143.166,Z 175.641,A -85,B 0,C 180,E1 -24333.436,E2 -24333.436} C_VEL
LIN {X 0,Y 143.129,Z 175.648,A -85,B 0,C 180,E1 -24339.666,E2 -24339.666} C_VEL
LIN {X 0,Y 143.18,Z 175.642,A -85,B 0,C 180,E1 -24343.406,E2 -24343.406} C_VEL
LIN {X 0,Y 143.168,Z 175.638,A -85,B 0,C 180,E1 -24347.418,E2 -24347.418} C_VEL
LIN {X 0,Y 143.166,Z 175.649,A -85,B 0,C 180,E1 -24351.759,E2 -24351.759} C_VEL
LIN {X 0,Y 143.186,Z 175.647,A -85,B 0,C 180,E1 -24357.324,E2 -24357.324} C_VEL
LIN {X 0,Y 143.188,Z 175.649,A -85,B 0,C 180,E1 -24362.062,E2 -24362.062} C_VEL
LIN {X 0,Y 143.272,Z 175.64,A -85,B 0,C 180,E1 -24368.746,E2 -24368.746} C_VEL
LIN {X 0,Y 143.313,Z 175.634,A -85,B 0,C 180,E1 -24372.89,E2 -24372.89} C_VEL
LIN {X 0,Y 143.599,Z 175.602,A -85,B 0,C 180,E1 -24378.712,E2 -24378.712} C_VEL
LIN {X 0,Y 143.664,Z 175.769,A -85,B 0,C 180,E1 -24380.365,E2 -24380.365} C_VEL
LIN {X 0,Y 144.749,Z 178.572,A -85,B 0,C 180,E1 -24380.883,E2 -24380.883} C_VEL
LIN {X 0,Y 146.187,Z 180.627,A -85,B 0,C 180,E1 -24381.437,E2 -24381.437} C_VEL
LIN {X 0,Y 155.828,Z 197.552,A -85,B 0,C 180,E1 -24385.062,E2 -24385.062} C_VEL
LIN {X 0,Y 165.216,Z 218.85,A -85,B 0,C 180,E1 -24388.383,E2 -24388.383} C_VEL
LIN {X 0,Y 165.83,Z 220.451,A -85,B 0,C 180,E1 -24388.601,E2 -24388.601} C_VEL
LIN {X 0,Y 162.344,Z 272.685,A -85,B 0,C 180,E1 -24391.021,E2 -24391.021} C_VEL
LIN {X 0,Y 160.778,Z 286.169,A -85,B 0,C 180,E1 -24392.116,E2 -24392.116} C_VEL
LIN {X 0,Y 158.92,Z 298.734,A -85,B 0,C 180,E1 -24393.646,E2 -24393.646} C_VEL
LIN {X 0,Y 156.608,Z 310.595,A -85,B 0,C 180,E1 -24395.602,E2 -24395.602} C_VEL
LIN {X 0,Y 153.958,Z 321.352,A -85,B 0,C 180,E1 -24397.873,E2 -24397.873} C_VEL
LIN {X 0,Y 151.163,Z 331.853,A -85,B 0,C 180,E1 -24400.719,E2 -24400.719} C_VEL
LIN {X 0,Y 148.726,Z 340.45,A -85,B 0,C 180,E1 -24403.668,E2 -24403.668} C_VEL
LIN {X 0,Y 146.116,Z 349.31,A -85,B 0,C 180,E1 -24407.496,E2 -24407.496} C_VEL
LIN {X 0,Y 143.846,Z 357.169,A -85,B 0,C 180,E1 -24411.833,E2 -24411.833} C_VEL
LIN {X 0,Y 142.169,Z 363.516,A -85,B 0,C 180,E1 -24416.419,E2 -24416.419} C_VEL
LIN {X 0,Y 141.245,Z 367.274,A -85,B 0,C 180,E1 -24419.842,E2 -24419.842} C_VEL
LIN {X 0,Y 140.426,Z 371.545,A -85,B 0,C 180,E1 -24425.046,E2 -24425.046} C_VEL
LIN {X 0,Y 140.488,Z 374.493,A -85,B 0,C 180,E1 -24430.569,E2 -24430.569} C_VEL
LIN {X 0,Y 141.426,Z 375.936,A -85,B 0,C 180,E1 -24435.918,E2 -24435.918} C_VEL
LIN {X 0,Y 143.535,Z 375.91,A -85,B 0,C 180,E1 -24441.577,E2 -24441.577} C_VEL
LIN {X 0,Y 145.508,Z 375.068,A -85,B 0,C 180,E1 -24445.198,E2 -24445.198} C_VEL
LIN {X 0,Y 149.4,Z 372.442,A -85,B 0,C 180,E1 -24450.493,E2 -24450.493} C_VEL
LIN {X 0,Y 154.482,Z 368.127,A -85,B 0,C 180,E1 -24455.492,E2 -24455.492} C_VEL
LIN {X 0,Y 159.456,Z 363.136,A -85,B 0,C 180,E1 -24459.355,E2 -24459.355} C_VEL
LIN {X 0,Y 164.46,Z 357.487,A -85,B 0,C 180,E1 -24462.596,E2 -24462.596} C_VEL
LIN {X 0,Y 169.995,Z 350.466,A -85,B 0,C 180,E1 -24465.639,E2 -24465.639} C_VEL
LIN {X 0,Y 175.893,Z 341.863,A -85,B 0,C 180,E1 -24468.477,E2 -24468.477} C_VEL
LIN {X 0,Y 181.697,Z 332.02,A -85,B 0,C 180,E1 -24470.893,E2 -24470.893} C_VEL
LIN {X 0,Y 186.683,Z 321.975,A -85,B 0,C 180,E1 -24472.81,E2 -24472.81} C_VEL
LIN {X 0,Y 191.49,Z 310.346,A -85,B 0,C 180,E1 -24474.503,E2 -24474.503} C_VEL
LIN {X 0,Y 195.498,Z 297.917,A -85,B 0,C 180,E1 -24475.878,E2 -24475.878} C_VEL
LIN {X 0,Y 198.634,Z 285.038,A -85,B 0,C 180,E1 -24476.904,E2 -24476.904} C_VEL
LIN {X 0,Y 200.713,Z 272.91,A -85,B 0,C 180,E1 -24477.506,E2 -24477.506} C_VEL
LIN {X 0,Y 203.273,Z 248.229,A -85,B 0,C 180,E1 -24478.432,E2 -24478.432} C_VEL
LIN {X 0,Y 200.159,Z 241.519,A -85,B 0,C 180,E1 -24481.1,E2 -24481.1} C_VEL
LIN {X 0,Y 196.281,Z 234.1,A -85,B 0,C 180,E1 -24485.172,E2 -24485.172} C_VEL
LIN {X 0,Y 195.379,Z 232.656,A -85,B 0,C 180,E1 -24486.318,E2 -24486.318} C_VEL
LIN {X 0,Y 193.234,Z 229.064,A -85,B 0,C 180,E1 -24489.585,E2 -24489.585} C_VEL
LIN {X 0,Y 191.061,Z 225.388,A -85,B 0,C 180,E1 -24495.778,E2 -24495.778} C_VEL
LIN {X 0,Y 190.741,Z 225.355,A -85,B 0,C 180,E1 -24498.16,E2 -24498.16} C_VEL
LIN {X 0,Y 191.226,Z 226.736,A -85,B 0,C 180,E1 -24503.05,E2 -24503.05} C_VEL
LIN {X 0,Y 193.769,Z 232.591,A -85,B 0,C 180,E1 -24509.136,E2 -24509.136} C_VEL
LIN {X 0,Y 195.833,Z 237.584,A -85,B 0,C 180,E1 -24512.235,E2 -24512.235} C_VEL
LIN {X 0,Y 198.115,Z 243.025,A -85,B 0,C 180,E1 -24514.872,E2 -24514.872} C_VEL
LIN {X 0,Y 200.493,Z 249.308,A -85,B 0,C 180,E1 -24517.279,E2 -24517.279} C_VEL
LIN {X 0,Y 202.725,Z 255.953,A -85,B 0,C 180,E1 -24519.299,E2 -24519.299} C_VEL
LIN {X 0,Y 199.493,Z 284.293,A -85,B 0,C 180,E1 -24520.304,E2 -24520.304} C_VEL
LIN {X 0,Y 197.08,Z 296.449,A -85,B 0,C 180,E1 -24520.948,E2 -24520.948} C_VEL
LIN {X 0,Y 193.576,Z 309.075,A -85,B 0,C 180,E1 -24521.901,E2 -24521.901} C_VEL
LIN {X 0,Y 189.739,Z 319.763,A -85,B 0,C 180,E1 -24522.982,E2 -24522.982} C_VEL
LIN {X 0,Y 184.21,Z 332.329,A -85,B 0,C 180,E1 -24524.716,E2 -24524.716} C_VEL
LIN {X 0,Y 178.864,Z 342.433,A -85,B 0,C 180,E1 -24526.556,E2 -24526.556} C_VEL
LIN {X 0,Y 173.303,Z 351.596,A -85,B 0,C 180,E1 -24528.775,E2 -24528.775} C_VEL
LIN {X 0,Y 168.123,Z 359.208,A -85,B 0,C 180,E1 -24531.166,E2 -24531.166} C_VEL
LIN {X 0,Y 162.345,Z 366.738,A -85,B 0,C 180,E1 -24534.236,E2 -24534.236} C_VEL
LIN {X 0,Y 157.166,Z 372.885,A -85,B 0,C 180,E1 -24537.545,E2 -24537.545} C_VEL
LIN {X 0,Y 152.547,Z 378.048,A -85,B 0,C 180,E1 -24541.294,E2 -24541.294} C_VEL
LIN {X 0,Y 147.712,Z 382.81,A -85,B 0,C 180,E1 -24546.143,E2 -24546.143} C_VEL
LIN {X 0,Y 144.778,Z 385.396,A -85,B 0,C 180,E1 -24550.133,E2 -24550.133} C_VEL
LIN {X 0,Y 143.197,Z 386.638,A -85,B 0,C 180,E1 -24552.872,E2 -24552.872} C_VEL
LIN {X 0,Y 141.333,Z 387.934,A -85,B 0,C 180,E1 -24558.473,E2 -24558.473} C_VEL
LIN {X 0,Y 140.316,Z 388.091,A -85,B 0,C 180,E1 -24560.838,E2 -24560.838} C_VEL
LIN {X 0,Y 138.631,Z 387.836,A -85,B 0,C 180,E1 -24563.173,E2 -24563.173} C_VEL
LIN {X 0,Y 135.003,Z 386.314,A -85,B 0,C 180,E1 -24567.918,E2 -24567.918} C_VEL
LIN {X 0,Y 133.819,Z 384.685,A -85,B 0,C 180,E1 -24571.218,E2 -24571.218} C_VEL
LIN {X 0,Y 133.764,Z 383.501,A -85,B 0,C 180,E1 -24573.348,E2 -24573.348} C_VEL
LIN {X 0,Y 133.829,Z 380.326,A -85,B 0,C 180,E1 -24577.542,E2 -24577.542} C_VEL
LIN {X 0,Y 134.414,Z 375.8,A -85,B 0,C 180,E1 -24582.071,E2 -24582.071} C_VEL
LIN {X 0,Y 135.982,Z 368.863,A -85,B 0,C 180,E1 -24587.287,E2 -24587.287} C_VEL
LIN {X 0,Y 138.149,Z 361.3,A -85,B 0,C 180,E1 -24591.641,E2 -24591.641} C_VEL
LIN {X 0,Y 140.744,Z 352.485,A -85,B 0,C 180,E1 -24595.6,E2 -24595.6} C_VEL
LIN {X 0,Y 143.589,Z 343.146,A -85,B 0,C 180,E1 -24598.862,E2 -24598.862} C_VEL
LIN {X 0,Y 146.302,Z 333.643,A -85,B 0,C 180,E1 -24601.492,E2 -24601.492} C_VEL
LIN {X 0,Y 149.344,Z 322.098,A -85,B 0,C 180,E1 -24603.973,E2 -24603.973} C_VEL
LIN {X 0,Y 151.971,Z 309.946,A -85,B 0,C 180,E1 -24605.924,E2 -24605.924} C_VEL
LIN {X 0,Y 154.218,Z 296.717,A -85,B 0,C 180,E1 -24607.45,E2 -24607.45} C_VEL
LIN {X 0,Y 155.843,Z 283.784,A -85,B 0,C 180,E1 -24608.423,E2 -24608.423} C_VEL
LIN {X 0,Y 158.5,Z 242.475,A -85,B 0,C 180,E1 -24610.428,E2 -24610.428} C_VEL
LIN {X 0,Y 156.862,Z 224.935,A -85,B 0,C 180,E1 -24611.839,E2 -24611.839} C_VEL
LIN {X 0,Y 149.839,Z 205.445,A -85,B 0,C 180,E1 -24614.746,E2 -24614.746} C_VEL
LIN {X 0,Y 143.399,Z 190.742,A -85,B 0,C 180,E1 -24617.498,E2 -24617.498} C_VEL
LIN {X 0,Y 139.989,Z 183.971,A -85,B 0,C 180,E1 -24619.002,E2 -24619.002} C_VEL
LIN {X 0,Y 137.828,Z 180.458,A -85,B 0,C 180,E1 -24619.951,E2 -24619.951} C_VEL
LIN {X 0,Y 136.301,Z 177.856,A -85,B 0,C 180,E1 -24620.654,E2 -24620.654} C_VEL
LIN {X 0,Y 136.015,Z 176.541,A -85,B 0,C 180,E1 -24620.901,E2 -24620.901} C_VEL
LIN {X 0,Y 136.056,Z 176.535,A -85,B 0,C 180,E1 -24625.736,E2 -24625.736} C_VEL
LIN {X 0,Y 136.147,Z 176.525,A -85,B 0,C 180,E1 -24632.315,E2 -24632.315} C_VEL
LIN {X 0,Y 136.234,Z 176.514,A -85,B 0,C 180,E1 -24638.83,E2 -24638.83} C_VEL
LIN {X 0,Y 136.252,Z 176.504,A -85,B 0,C 180,E1 -24645.053,E2 -24645.053} C_VEL
LIN {X 0,Y 136.495,Z 176.482,A -85,B 0,C 180,E1 -24648.113,E2 -24648.113} C_VEL
LIN {X 0,Y 136.587,Z 176.456,A -85,B 0,C 180,E1 -24651.119,E2 -24651.119} C_VEL
LIN {X 0,Y 137.133,Z 176.392,A -85,B 0,C 180,E1 -24659.998,E2 -24659.998} C_VEL
LIN {X 0,Y 136.589,Z 176.469,A -85,B 0,C 180,E1 -24668.878,E2 -24668.878} C_VEL
LIN {X 0,Y 136.487,Z 176.465,A -85,B 0,C 180,E1 -24671.953,E2 -24671.953} C_VEL
LIN {X 0,Y 136.249,Z 176.508,A -85,B 0,C 180,E1 -24678.027,E2 -24678.027} C_VEL
LIN {X 0,Y 136.195,Z 176.514,A -85,B 0,C 180,E1 -24681.749,E2 -24681.749} C_VEL
LIN {X 0,Y 136.096,Z 176.52,A -85,B 0,C 180,E1 -24688.616,E2 -24688.616} C_VEL
LIN {X 0,Y 136.079,Z 176.516,A -85,B 0,C 180,E1 -24694.617,E2 -24694.617} C_VEL
LIN {X 0,Y 136.102,Z 176.522,A -85,B 0,C 180,E1 -24699.237,E2 -24699.237} C_VEL
LIN {X 0,Y 136.115,Z 176.52,A -85,B 0,C 180,E1 -24703.711,E2 -24703.711} C_VEL
LIN {X 0,Y 136.115,Z 176.518,A -85,B 0,C 180,E1 -24707.84,E2 -24707.84} C_VEL
LIN {X 0,Y 136.117,Z 176.527,A -85,B 0,C 180,E1 -24711.716,E2 -24711.716} C_VEL
LIN {X 0,Y 136.09,Z 176.521,A -85,B 0,C 180,E1 -24715.715,E2 -24715.715} C_VEL
LIN {X 0,Y 136.143,Z 176.526,A -85,B 0,C 180,E1 -24722.318,E2 -24722.318} C_VEL
LIN {X 0,Y 136.239,Z 176.516,A -85,B 0,C 180,E1 -24728.834,E2 -24728.834} C_VEL
LIN {X 0,Y 136.282,Z 176.512,A -85,B 0,C 180,E1 -24735.059,E2 -24735.059} C_VEL
LIN {X 0,Y 136.525,Z 176.515,A -85,B 0,C 180,E1 -24738.171,E2 -24738.171} C_VEL
LIN {X 0,Y 137.586,Z 179.378,A -85,B 0,C 180,E1 -24738.744,E2 -24738.744} C_VEL
LIN {X 0,Y 139.225,Z 181.675,A -85,B 0,C 180,E1 -24739.446,E2 -24739.446} C_VEL
LIN {X 0,Y 145.323,Z 192.132,A -85,B 0,C 180,E1 -24742.006,E2 -24742.006} C_VEL
LIN {X 0,Y 150.86,Z 202.014,A -85,B 0,C 180,E1 -24744.131,E2 -24744.131} C_VEL
LIN {X 0,Y 159.501,Z 221.97,A -85,B 0,C 180,E1 -24747.397,E2 -24747.397} C_VEL
LIN {X 0,Y 156.037,Z 272.838,A -85,B 0,C 180,E1 -24749.848,E2 -24749.848} C_VEL
LIN {X 0,Y 154.462,Z 286.083,A -85,B 0,C 180,E1 -24750.952,E2 -24750.952} C_VEL
LIN {X 0,Y 152.551,Z 298.575,A -85,B 0,C 180,E1 -24752.502,E2 -24752.502} C_VEL
LIN {X 0,Y 150.326,Z 309.692,A -85,B 0,C 180,E1 -24754.359,E2 -24754.359} C_VEL
LIN {X 0,Y 147.214,Z 321.993,A -85,B 0,C 180,E1 -24757.03,E2 -24757.03} C_VEL
LIN {X 0,Y 144.205,Z 332.87,A -85,B 0,C 180,E1 -24760.146,E2 -24760.146} C_VEL
LIN {X 0,Y 141.319,Z 342.421,A -85,B 0,C 180,E1 -24763.665,E2 -24763.665} C_VEL
LIN {X 0,Y 138.713,Z 351.021,A -85,B 0,C 180,E1 -24767.7,E2 -24767.7} C_VEL
LIN {X 0,Y 136.53,Z 358.309,A -85,B 0,C 180,E1 -24772.099,E2 -24772.099} C_VEL
LIN {X 0,Y 135.159,Z 363.434,A -85,B 0,C 180,E1 -24775.995,E2 -24775.995} C_VEL
LIN {X 0,Y 134.137,Z 367.497,A -85,B 0,C 180,E1 -24779.853,E2 -24779.853} C_VEL
LIN {X 0,Y 133.591,Z 369.926,A -85,B 0,C 180,E1 -24782.68,E2 -24782.68} C_VEL
LIN {X 0,Y 133.218,Z 373.207,A -85,B 0,C 180,E1 -24787.693,E2 -24787.693} C_VEL
LIN {X 0,Y 133.695,Z 375.441,A -85,B 0,C 180,E1 -24793.111,E2 -24793.111} C_VEL
LIN {X 0,Y 134.691,Z 376.314,A -85,B 0,C 180,E1 -24797.29,E2 -24797.29} C_VEL
LIN {X 0,Y 136.432,Z 376.398,A -85,B 0,C 180,E1 -24801.821,E2 -24801.821} C_VEL
LIN {X 0,Y 138.812,Z 375.579,A -85,B 0,C 180,E1 -24806.159,E2 -24806.159} C_VEL
LIN {X 0,Y 141.816,Z 373.873,A -85,B 0,C 180,E1 -24810.295,E2 -24810.295} C_VEL
LIN {X 0,Y 146.812,Z 370.24,A -85,B 0,C 180,E1 -24815.446,E2 -24815.446} C_VEL
LIN {X 0,Y 152.66,Z 365.067,A -85,B 0,C 180,E1 -24820.126,E2 -24820.126} C_VEL
LIN {X 0,Y 158.783,Z 358.768,A -85,B 0,C 180,E1 -24824.031,E2 -24824.031} C_VEL
LIN {X 0,Y 165.507,Z 350.719,A -85,B 0,C 180,E1 -24827.604,E2 -24827.604} C_VEL
LIN {X 0,Y 171.176,Z 342.893,A -85,B 0,C 180,E1 -24830.196,E2 -24830.196} C_VEL
LIN {X 0,Y 177.187,Z 333.38,A -85,B 0,C 180,E1 -24832.582,E2 -24832.582} C_VEL
LIN {X 0,Y 182.803,Z 322.713,A -85,B 0,C 180,E1 -24834.645,E2 -24834.645} C_VEL
LIN {X 0,Y 187.958,Z 310.853,A -85,B 0,C 180,E1 -24836.367,E2 -24836.367} C_VEL
LIN {X 0,Y 191.879,Z 299.306,A -85,B 0,C 180,E1 -24837.64,E2 -24837.64} C_VEL
LIN {X 0,Y 195.332,Z 285.887,A -85,B 0,C 180,E1 -24838.712,E2 -24838.712} C_VEL
LIN {X 0,Y 197.516,Z 273.864,A -85,B 0,C 180,E1 -24839.31,E2 -24839.31} C_VEL
LIN {X 0,Y 199.908,Z 251.973,A -85,B 0,C 180,E1 -24840.124,E2 -24840.124} C_VEL
LIN {X 0,Y 197.498,Z 246.5,A -85,B 0,C 180,E1 -24842.488,E2 -24842.488} C_VEL
LIN {X 0,Y 194.238,Z 239.814,A -85,B 0,C 180,E1 -24846.355,E2 -24846.355} C_VEL
LIN {X 0,Y 191.859,Z 235.865,A -85,B 0,C 180,E1 -24850.122,E2 -24850.122} C_VEL
LIN {X 0,Y 189.979,Z 232.474,A -85,B 0,C 180,E1 -24855.876,E2 -24855.876} C_VEL
LIN {X 0,Y 189.669,Z 232.464,A -85,B 0,C 180,E1 -24858.784,E2 -24858.784} C_VEL
LIN {X 0,Y 190.127,Z 233.804,A -85,B 0,C 180,E1 -24862.918,E2 -24862.918} C_VEL
LIN {X 0,Y 192.24,Z 239.174,A -85,B 0,C 180,E1 -24868.474,E2 -24868.474} C_VEL
LIN {X 0,Y 194.111,Z 244.098,A -85,B 0,C 180,E1 -24871.527,E2 -24871.527} C_VEL
LIN {X 0,Y 195.919,Z 248.775,A -85,B 0,C 180,E1 -24873.837,E2 -24873.837} C_VEL
LIN {X 0,Y 198.114,Z 255.162,A -85,B 0,C 180,E1 -24876.32,E2 -24876.32} C_VEL
LIN {X 0,Y 199.361,Z 259.055,A -85,B 0,C 180,E1 -24877.566,E2 -24877.566} C_VEL
LIN {X 0,Y 196.414,Z 283.856,A -85,B 0,C 180,E1 -24878.441,E2 -24878.441} C_VEL
LIN {X 0,Y 193.775,Z 296.687,A -85,B 0,C 180,E1 -24879.114,E2 -24879.114} C_VEL
LIN {X 0,Y 190.338,Z 308.563,A -85,B 0,C 180,E1 -24879.987,E2 -24879.987} C_VEL
LIN {X 0,Y 186.369,Z 319.241,A -85,B 0,C 180,E1 -24881.042,E2 -24881.042} C_VEL
LIN {X 0,Y 180.63,Z 331.775,A -85,B 0,C 180,E1 -24882.742,E2 -24882.742} C_VEL
LIN {X 0,Y 175.045,Z 341.869,A -85,B 0,C 180,E1 -24884.547,E2 -24884.547} C_VEL
LIN {X 0,Y 169.225,Z 351.065,A -85,B 0,C 180,E1 -24886.742,E2 -24886.742} C_VEL
LIN {X 0,Y 163.649,Z 358.731,A -85,B 0,C 180,E1 -24889.084,E2 -24889.084} C_VEL
LIN {X 0,Y 157.667,Z 366.268,A -85,B 0,C 180,E1 -24892.198,E2 -24892.198} C_VEL
LIN {X 0,Y 151.242,Z 373.331,A -85,B 0,C 180,E1 -24896.107,E2 -24896.107} C_VEL
LIN {X 0,Y 147.079,Z 377.584,A -85,B 0,C 180,E1 -24899.332,E2 -24899.332} C_VEL
LIN {X 0,Y 142.443,Z 381.817,A -85,B 0,C 180,E1 -24903.636,E2 -24903.636} C_VEL
LIN {X 0,Y 140.113,Z 383.787,A -85,B 0,C 180,E1 -24906.34,E2 -24906.34} C_VEL
LIN {X 0,Y 138.099,Z 385.336,A -85,B 0,C 180,E1 -24909.129,E2 -24909.129} C_VEL
LIN {X 0,Y 136.397,Z 386.472,A -85,B 0,C 180,E1 -24911.99,E2 -24911.99} C_VEL
LIN {X 0,Y 134.332,Z 387.642,A -85,B 0,C 180,E1 -24917.919,E2 -24917.919} C_VEL
LIN {X 0,Y 133.8,Z 387.674,A -85,B 0,C 180,E1 -24920.932,E2 -24920.932} C_VEL
LIN {X 0,Y 133.609,Z 387.3,A -85,B 0,C 180,E1 -24923.959,E2 -24923.959} C_VEL
LIN {X 0,Y 133.69,Z 386.438,A -85,B 0,C 180,E1 -24927.241,E2 -24927.241} C_VEL
LIN {X 0,Y 133.933,Z 385.35,A -85,B 0,C 180,E1 -24929.998,E2 -24929.998} C_VEL
LIN {X 0,Y 133.819,Z 384.685,A -85,B 0,C 180,E1 -24931.218,E2 -24931.218} C_VEL
LIN {X 0,Y 133.044,Z 383.238,A -85,B 0,C 180,E1 -24933.644,E2 -24933.644} C_VEL
LIN {X 0,Y 131.48,Z 381.425,A -85,B 0,C 180,E1 -24936.005,E2 -24936.005} C_VEL
LIN {X 0,Y 128.205,Z 376.992,A -85,B 0,C 180,E1 -24940.714,E2 -24940.714} C_VEL
LIN {X 0,Y 127.613,Z 374.388,A -85,B 0,C 180,E1 -24943.112,E2 -24943.112} C_VEL
LIN {X 0,Y 127.718,Z 373.456,A -85,B 0,C 180,E1 -24943.907,E2 -24943.907} C_VEL
LIN {X 0,Y 129.539,Z 366.522,A -85,B 0,C 180,E1 -24948.995,E2 -24948.995} C_VEL
LIN {X 0,Y 131.95,Z 358.398,A -85,B 0,C 180,E1 -24953.543,E2 -24953.543} C_VEL
LIN {X 0,Y 134.546,Z 350.249,A -85,B 0,C 180,E1 -24957.131,E2 -24957.131} C_VEL
LIN {X 0,Y 137.773,Z 339.998,A -85,B 0,C 180,E1 -24960.67,E2 -24960.67} C_VEL
LIN {X 0,Y 140.615,Z 329.966,A -85,B 0,C 180,E1 -24963.35,E2 -24963.35} C_VEL
LIN {X 0,Y 143.891,Z 317.435,A -85,B 0,C 180,E1 -24965.88,E2 -24965.88} C_VEL
LIN {X 0,Y 146.504,Z 305.112,A -85,B 0,C 180,E1 -24967.706,E2 -24967.706} C_VEL
LIN {X 0,Y 148.608,Z 291.423,A -85,B 0,C 180,E1 -24969.126,E2 -24969.126} C_VEL
LIN {X 0,Y 149.932,Z 279.391,A -85,B 0,C 180,E1 -24969.909,E2 -24969.909} C_VEL
LIN {X 0,Y 152.32,Z 243.001,A -85,B 0,C 180,E1 -24971.708,E2 -24971.708} C_VEL
LIN {X 0,Y 150.889,Z 227.144,A -85,B 0,C 180,E1 -24973.054,E2 -24973.054} C_VEL
LIN {X 0,Y 144.439,Z 208.94,A -85,B 0,C 180,E1 -24975.923,E2 -24975.923} C_VEL
LIN {X 0,Y 138.114,Z 194.254,A -85,B 0,C 180,E1 -24978.806,E2 -24978.806} C_VEL
LIN {X 0,Y 134.453,Z 187.094,A -85,B 0,C 180,E1 -24980.547,E2 -24980.547} C_VEL
LIN {X 0,Y 131.65,Z 182.505,A -85,B 0,C 180,E1 -24981.882,E2 -24981.882} C_VEL
LIN {X 0,Y 129.434,Z 179.258,A -85,B 0,C 180,E1 -24982.958,E2 -24982.958} C_VEL
LIN {X 0,Y 128.94,Z 177.428,A -85,B 0,C 180,E1 -24983.402,E2 -24983.402} C_VEL
LIN {X 0,Y 128.978,Z 177.42,A -85,B 0,C 180,E1 -24986.98,E2 -24986.98} C_VEL
LIN {X 0,Y 129.05,Z 177.401,A -85,B 0,C 180,E1 -24990.649,E2 -24990.649} C_VEL
LIN {X 0,Y 129.104,Z 177.396,A -85,B 0,C 180,E1 -24997.727,E2 -24997.727} C_VEL
LIN {X 0,Y 129.169,Z 177.382,A -85,B 0,C 180,E1 -25004.212,E2 -25004.212} C_VEL
LIN {X 0,Y 129.414,Z 177.365,A -85,B 0,C 180,E1 -25007.818,E2 -25007.818} C_VEL
LIN {X 0,Y 129.513,Z 177.339,A -85,B 0,C 180,E1 -25010.629,E2 -25010.629} C_VEL
LIN {X 0,Y 130.088,Z 177.269,A -85,B 0,C 180,E1 -25019.998,E2 -25019.998} C_VEL
LIN {X 0,Y 129.514,Z 177.349,A -85,B 0,C 180,E1 -25029.367,E2 -25029.367} C_VEL
LIN {X 0,Y 129.39,Z 177.344,A -85,B 0,C 180,E1 -25032.547,E2 -25032.547} C_VEL
LIN {X 0,Y 129.157,Z 177.395,A -85,B 0,C 180,E1 -25039.054,E2 -25039.054} C_VEL
LIN {X 0,Y 129.104,Z 177.392,A -85,B 0,C 180,E1 -25042.397,E2 -25042.397} C_VEL
LIN {X 0,Y 129.031,Z 177.404,A -85,B 0,C 180,E1 -25049.372,E2 -25049.372} C_VEL
LIN {X 0,Y 129.024,Z 177.389,A -85,B 0,C 180,E1 -25055.212,E2 -25055.212} C_VEL
LIN {X 0,Y 129.046,Z 177.406,A -85,B 0,C 180,E1 -25060.806,E2 -25060.806} C_VEL
LIN {X 0,Y 129.036,Z 177.394,A -85,B 0,C 180,E1 -25065.074,E2 -25065.074} C_VEL
LIN {X 0,Y 129.046,Z 177.408,A -85,B 0,C 180,E1 -25069.678,E2 -25069.678} C_VEL
LIN {X 0,Y 129.025,Z 177.398,A -85,B 0,C 180,E1 -25074.788,E2 -25074.788} C_VEL
LIN {X 0,Y 129.046,Z 177.408,A -85,B 0,C 180,E1 -25080.652,E2 -25080.652} C_VEL
LIN {X 0,Y 129.103,Z 177.404,A -85,B 0,C 180,E1 -25087.729,E2 -25087.729} C_VEL
LIN {X 0,Y 129.156,Z 177.399,A -85,B 0,C 180,E1 -25090.946,E2 -25090.946} C_VEL
LIN {X 0,Y 129.25,Z 177.388,A -85,B 0,C 180,E1 -25095.678,E2 -25095.678} C_VEL
LIN {X 0,Y 130.219,Z 180.104,A -85,B 0,C 180,E1 -25096.273,E2 -25096.273} C_VEL
LIN {X 0,Y 132.317,Z 182.756,A -85,B 0,C 180,E1 -25097.232,E2 -25097.232} C_VEL
LIN {X 0,Y 138.352,Z 192.781,A -85,B 0,C 180,E1 -25100.013,E2 -25100.013} C_VEL
LIN {X 0,Y 145.498,Z 205.686,A -85,B 0,C 180,E1 -25102.995,E2 -25102.995} C_VEL
LIN {X 0,Y 153.323,Z 223.823,A -85,B 0,C 180,E1 -25106.146,E2 -25106.146} C_VEL
LIN {X 0,Y 149.784,Z 273.129,A -85,B 0,C 180,E1 -25108.589,E2 -25108.589} C_VEL
LIN {X 0,Y 148.148,Z 286.517,A -85,B 0,C 180,E1 -25109.747,E2 -25109.747} C_VEL
LIN {X 0,Y 146.277,Z 298.25,A -85,B 0,C 180,E1 -25111.24,E2 -25111.24} C_VEL
LIN {X 0,Y 143.961,Z 309.49,A -85,B 0,C 180,E1 -25113.15,E2 -25113.15} C_VEL
LIN {X 0,Y 140.907,Z 321.142,A -85,B 0,C 180,E1 -25115.727,E2 -25115.727} C_VEL
LIN {X 0,Y 137.817,Z 331.825,A -85,B 0,C 180,E1 -25118.802,E2 -25118.802} C_VEL
LIN {X 0,Y 135.171,Z 340.545,A -85,B 0,C 180,E1 -25122.005,E2 -25122.005} C_VEL
LIN {X 0,Y 132.395,Z 349.149,A -85,B 0,C 180,E1 -25125.997,E2 -25125.997} C_VEL
LIN {X 0,Y 129.999,Z 356.861,A -85,B 0,C 180,E1 -25130.575,E2 -25130.575} C_VEL
LIN {X 0,Y 128.264,Z 362.848,A -85,B 0,C 180,E1 -25135.13,E2 -25135.13} C_VEL
LIN {X 0,Y 127.003,Z 367.701,A -85,B 0,C 180,E1 -25139.872,E2 -25139.872} C_VEL
LIN {X 0,Y 126.181,Z 372.13,A -85,B 0,C 180,E1 -25145.793,E2 -25145.793} C_VEL
LIN {X 0,Y 126.394,Z 375.08,A -85,B 0,C 180,E1 -25151.857,E2 -25151.857} C_VEL
LIN {X 0,Y 127.16,Z 376.258,A -85,B 0,C 180,E1 -25155.933,E2 -25155.933} C_VEL
LIN {X 0,Y 128.465,Z 376.789,A -85,B 0,C 180,E1 -25159.991,E2 -25159.991} C_VEL
LIN {X 0,Y 130.283,Z 376.646,A -85,B 0,C 180,E1 -25164.017,E2 -25164.017} C_VEL
LIN {X 0,Y 132.715,Z 375.843,A -85,B 0,C 180,E1 -25168.026,E2 -25168.026} C_VEL
LIN {X 0,Y 136.037,Z 374.11,A -85,B 0,C 180,E1 -25172.294,E2 -25172.294} C_VEL
LIN {X 0,Y 141.458,Z 370.444,A -85,B 0,C 180,E1 -25177.526,E2 -25177.526} C_VEL
LIN {X 0,Y 147.654,Z 365.34,A -85,B 0,C 180,E1 -25182.173,E2 -25182.173} C_VEL
LIN {X 0,Y 154.189,Z 359.003,A -85,B 0,C 180,E1 -25186.105,E2 -25186.105} C_VEL
LIN {X 0,Y 160.764,Z 351.608,A -85,B 0,C 180,E1 -25189.441,E2 -25189.441} C_VEL
LIN {X 0,Y 166.761,Z 343.852,A -85,B 0,C 180,E1 -25192.059,E2 -25192.059} C_VEL
LIN {X 0,Y 173.013,Z 334.565,A -85,B 0,C 180,E1 -25194.411,E2 -25194.411} C_VEL
LIN {X 0,Y 178.69,Z 324.361,A -85,B 0,C 180,E1 -25196.41,E2 -25196.41} C_VEL
LIN {X 0,Y 184.101,Z 312.645,A -85,B 0,C 180,E1 -25198.138,E2 -25198.138} C_VEL
LIN {X 0,Y 188.45,Z 300.766,A -85,B 0,C 180,E1 -25199.461,E2 -25199.461} C_VEL
LIN {X 0,Y 192.074,Z 287.678,A -85,B 0,C 180,E1 -25200.512,E2 -25200.512} C_VEL
LIN {X 0,Y 194.589,Z 274.813,A -85,B 0,C 180,E1 -25201.183,E2 -25201.183} C_VEL
LIN {X 0,Y 196.8,Z 255.808,A -85,B 0,C 180,E1 -25201.891,E2 -25201.891} C_VEL
LIN {X 0,Y 195.036,Z 251.915,A -85,B 0,C 180,E1 -25203.791,E2 -25203.791} C_VEL
LIN {X 0,Y 192.581,Z 246.298,A -85,B 0,C 180,E1 -25207.077,E2 -25207.077} C_VEL
LIN {X 0,Y 190.521,Z 242.676,A -85,B 0,C 180,E1 -25210.63,E2 -25210.63} C_VEL
LIN {X 0,Y 188.848,Z 239.433,A -85,B 0,C 180,E1 -25216.347,E2 -25216.347} C_VEL
LIN {X 0,Y 188.641,Z 239.673,A -85,B 0,C 180,E1 -25219.592,E2 -25219.592} C_VEL
LIN {X 0,Y 189.008,Z 240.882,A -85,B 0,C 180,E1 -25222.71,E2 -25222.71} C_VEL
LIN {X 0,Y 190.751,Z 245.826,A -85,B 0,C 180,E1 -25227.838,E2 -25227.838} C_VEL
LIN {X 0,Y 192.403,Z 250.51,A -85,B 0,C 180,E1 -25230.757,E2 -25230.757} C_VEL
LIN {X 0,Y 194.182,Z 255.607,A -85,B 0,C 180,E1 -25233.276,E2 -25233.276} C_VEL
LIN {X 0,Y 196.208,Z 262.297,A -85,B 0,C 180,E1 -25235.754,E2 -25235.754} C_VEL
LIN {X 0,Y 193.537,Z 283.673,A -85,B 0,C 180,E1 -25236.532,E2 -25236.532} C_VEL
LIN {X 0,Y 190.661,Z 296.967,A -85,B 0,C 180,E1 -25237.217,E2 -25237.217} C_VEL
LIN {X 0,Y 186.629,Z 309.971,A -85,B 0,C 180,E1 -25238.175,E2 -25238.175} C_VEL
LIN {X 0,Y 181.89,Z 321.813,A -85,B 0,C 180,E1 -25239.394,E2 -25239.394} C_VEL
LIN {X 0,Y 176.632,Z 332.586,A -85,B 0,C 180,E1 -25240.886,E2 -25240.886} C_VEL
LIN {X 0,Y 170.211,Z 343.417,A -85,B 0,C 180,E1 -25242.868,E2 -25242.868} C_VEL
LIN {X 0,Y 163.008,Z 353.849,A -85,B 0,C 180,E1 -25245.522,E2 -25245.522} C_VEL
LIN {X 0,Y 157.408,Z 360.941,A -85,B 0,C 180,E1 -25247.952,E2 -25247.952} C_VEL
LIN {X 0,Y 151.138,Z 368.032,A -85,B 0,C 180,E1 -25251.113,E2 -25251.113} C_VEL
LIN {X 0,Y 145.432,Z 373.785,A -85,B 0,C 180,E1 -25254.554,E2 -25254.554} C_VEL
LIN {X 0,Y 140.665,Z 378.208,A -85,B 0,C 180,E1 -25258.145,E2 -25258.145} C_VEL
LIN {X 0,Y 136.12,Z 381.946,A -85,B 0,C 180,E1 -25262.309,E2 -25262.309} C_VEL
LIN {X 0,Y 131.47,Z 385.236,A -85,B 0,C 180,E1 -25268.023,E2 -25268.023} C_VEL
LIN {X 0,Y 128.314,Z 387.01,A -85,B 0,C 180,E1 -25274.104,E2 -25274.104} C_VEL
LIN {X 0,Y 127.37,Z 387.34,A -85,B 0,C 180,E1 -25277.247,E2 -25277.247} C_VEL
LIN {X 0,Y 126.536,Z 386.809,A -85,B 0,C 180,E1 -25283.62,E2 -25283.62} C_VEL
LIN {X 0,Y 126.639,Z 385.796,A -85,B 0,C 180,E1 -25287.391,E2 -25287.391} C_VEL
LIN {X 0,Y 126.853,Z 384.747,A -85,B 0,C 180,E1 -25289.998,E2 -25289.998} C_VEL
LIN {X 0,Y 126.628,Z 381.949,A -85,B 0,C 180,E1 -25294.774,E2 -25294.774} C_VEL
LIN {X 0,Y 126.965,Z 378.065,A -85,B 0,C 180,E1 -25299.557,E2 -25299.557} C_VEL
LIN {X 0,Y 127.718,Z 373.456,A -85,B 0,C 180,E1 -25303.907,E2 -25303.907} C_VEL
LIN {X 0,Y 127.721,Z 370.57,A -85,B 0,C 180,E1 -25306.223,E2 -25306.223} C_VEL
LIN {X 0,Y 126.312,Z 365.239,A -85,B 0,C 180,E1 -25309.948,E2 -25309.948} C_VEL
LIN {X 0,Y 125.287,Z 359.315,A -85,B 0,C 180,E1 -25313.555,E2 -25313.555} C_VEL
LIN {X 0,Y 125.89,Z 355.405,A -85,B 0,C 180,E1 -25315.588,E2 -25315.588} C_VEL
LIN {X 0,Y 128.942,Z 346.457,A -85,B 0,C 180,E1 -25319.374,E2 -25319.374} C_VEL
LIN {X 0,Y 132.454,Z 335.544,A -85,B 0,C 180,E1 -25322.945,E2 -25322.945} C_VEL
LIN {X 0,Y 135.565,Z 324.53,A -85,B 0,C 180,E1 -25325.676,E2 -25325.676} C_VEL
LIN {X 0,Y 138.62,Z 312.342,A -85,B 0,C 180,E1 -25327.931,E2 -25327.931} C_VEL
LIN {X 0,Y 140.883,Z 300.953,A -85,B 0,C 180,E1 -25329.495,E2 -25329.495} C_VEL
LIN {X 0,Y 142.839,Z 288.256,A -85,B 0,C 180,E1 -25330.696,E2 -25330.696} C_VEL
LIN {X 0,Y 144.291,Z 271.805,A -85,B 0,C 180,E1 -25331.656,E2 -25331.656} C_VEL
LIN {X 0,Y 146.205,Z 243.423,A -85,B 0,C 180,E1 -25333.108,E2 -25333.108} C_VEL
LIN {X 0,Y 144.919,Z 229.17,A -85,B 0,C 180,E1 -25334.403,E2 -25334.403} C_VEL
LIN {X 0,Y 138.843,Z 211.808,A -85,B 0,C 180,E1 -25337.273,E2 -25337.273} C_VEL
LIN {X 0,Y 132.367,Z 196.523,A -85,B 0,C 180,E1 -25340.501,E2 -25340.501} C_VEL
LIN {X 0,Y 129.076,Z 190.452,A -85,B 0,C 180,E1 -25342.147,E2 -25342.147} C_VEL
LIN {X 0,Y 124.6,Z 183.193,A -85,B 0,C 180,E1 -25344.482,E2 -25344.482} C_VEL
LIN {X 0,Y 122.491,Z 180.339,A -85,B 0,C 180,E1 -25345.61,E2 -25345.61} C_VEL
LIN {X 0,Y 121.924,Z 178.295,A -85,B 0,C 180,E1 -25346.114,E2 -25346.114} C_VEL
LIN {X 0,Y 121.956,Z 178.293,A -85,B 0,C 180,E1 -25352.545,E2 -25352.545} C_VEL
LIN {X 0,Y 122.021,Z 178.275,A -85,B 0,C 180,E1 -25357.149,E2 -25357.149} C_VEL
LIN {X 0,Y 122.082,Z 178.263,A -85,B 0,C 180,E1 -25363.269,E2 -25363.269} C_VEL
LIN {X 0,Y 122.328,Z 178.248,A -85,B 0,C 180,E1 -25367.594,E2 -25367.594} C_VEL
LIN {X 0,Y 122.443,Z 178.223,A -85,B 0,C 180,E1 -25370.083,E2 -25370.083} C_VEL
LIN {X 0,Y 122.605,Z 178.212,A -85,B 0,C 180,E1 -25376.712,E2 -25376.712} C_VEL
LIN {X 0,Y 123.041,Z 178.146,A -85,B 0,C 180,E1 -25379.998,E2 -25379.998} C_VEL
LIN {X 0,Y 122.416,Z 178.23,A -85,B 0,C 180,E1 -25387.121,E2 -25387.121} C_VEL
LIN {X 0,Y 122.36,Z 178.219,A -85,B 0,C 180,E1 -25392.472,E2 -25392.472} C_VEL
LIN {X 0,Y 122.114,Z 178.262,A -85,B 0,C 180,E1 -25396.722,E2 -25396.722} C_VEL
LIN {X 0,Y 122.019,Z 178.271,A -85,B 0,C 180,E1 -25402.85,E2 -25402.85} C_VEL
LIN {X 0,Y 121.945,Z 178.273,A -85,B 0,C 180,E1 -25407.453,E2 -25407.453} C_VEL
LIN {X 0,Y 121.908,Z 178.294,A -85,B 0,C 180,E1 -25411.253,E2 -25411.253} C_VEL
LIN {X 0,Y 121.946,Z 178.267,A -85,B 0,C 180,E1 -25416.214,E2 -25416.214} C_VEL
LIN {X 0,Y 121.965,Z 178.288,A -85,B 0,C 180,E1 -25421.491,E2 -25421.491} C_VEL
LIN {X 0,Y 121.965,Z 178.283,A -85,B 0,C 180,E1 -25428.509,E2 -25428.509} C_VEL
LIN {X 0,Y 121.976,Z 178.275,A -85,B 0,C 180,E1 -25434.82,E2 -25434.82} C_VEL
LIN {X 0,Y 121.938,Z 178.294,A -85,B 0,C 180,E1 -25439.826,E2 -25439.826} C_VEL
LIN {X 0,Y 121.979,Z 178.29,A -85,B 0,C 180,E1 -25446.216,E2 -25446.216} C_VEL
LIN {X 0,Y 122.092,Z 178.277,A -85,B 0,C 180,E1 -25452.412,E2 -25452.412} C_VEL
LIN {X 0,Y 122.087,Z 178.278,A -85,B 0,C 180,E1 -25452.843,E2 -25452.843} C_VEL
LIN {X 0,Y 123.225,Z 181.252,A -85,B 0,C 180,E1 -25453.635,E2 -25453.635} C_VEL
LIN {X 0,Y 125.081,Z 183.495,A -85,B 0,C 180,E1 -25454.602,E2 -25454.602} C_VEL
LIN {X 0,Y 127.092,Z 186.673,A -85,B 0,C 180,E1 -25455.667,E2 -25455.667} C_VEL
LIN {X 0,Y 131.948,Z 194.251,A -85,B 0,C 180,E1 -25458.038,E2 -25458.038} C_VEL
LIN {X 0,Y 140.29,Z 209.511,A -85,B 0,C 180,E1 -25461.83,E2 -25461.83} C_VEL
LIN {X 0,Y 147.205,Z 225.738,A -85,B 0,C 180,E1 -25464.793,E2 -25464.793} C_VEL
LIN {X 0,Y 143.645,Z 272.987,A -85,B 0,C 180,E1 -25467.197,E2 -25467.197} C_VEL
LIN {X 0,Y 141.949,Z 286.541,A -85,B 0,C 180,E1 -25468.399,E2 -25468.399} C_VEL
LIN {X 0,Y 139.886,Z 298.772,A -85,B 0,C 180,E1 -25470.002,E2 -25470.002} C_VEL
LIN {X 0,Y 137.197,Z 311.013,A -85,B 0,C 180,E1 -25472.204,E2 -25472.204} C_VEL
LIN {X 0,Y 134.022,Z 322.543,A -85,B 0,C 180,E1 -25474.92,E2 -25474.92} C_VEL
LIN {X 0,Y 130.902,Z 332.888,A -85,B 0,C 180,E1 -25478.104,E2 -25478.104} C_VEL
LIN {X 0,Y 127.559,Z 343.068,A -85,B 0,C 180,E1 -25482.189,E2 -25482.189} C_VEL
LIN {X 0,Y 124.707,Z 351.699,A -85,B 0,C 180,E1 -25486.66,E2 -25486.66} C_VEL
LIN {X 0,Y 122.43,Z 358.768,A -85,B 0,C 180,E1 -25491.384,E2 -25491.384} C_VEL
LIN {X 0,Y 120.611,Z 365.053,A -85,B 0,C 180,E1 -25496.848,E2 -25496.848} C_VEL
LIN {X 0,Y 119.486,Z 369.535,A -85,B 0,C 180,E1 -25501.965,E2 -25501.965} C_VEL
LIN {X 0,Y 119.059,Z 372.374,A -85,B 0,C 180,E1 -25506.18,E2 -25506.18} C_VEL
LIN {X 0,Y 119.151,Z 374.534,A -85,B 0,C 180,E1 -25510.456,E2 -25510.456} C_VEL
LIN {X 0,Y 119.878,Z 376.186,A -85,B 0,C 180,E1 -25515.293,E2 -25515.293} C_VEL
LIN {X 0,Y 121.462,Z 377.066,A -85,B 0,C 180,E1 -25520.473,E2 -25520.473} C_VEL
LIN {X 0,Y 123.753,Z 377.025,A -85,B 0,C 180,E1 -25525.398,E2 -25525.398} C_VEL
LIN {X 0,Y 127.897,Z 375.621,A -85,B 0,C 180,E1 -25531.551,E2 -25531.551} C_VEL
LIN {X 0,Y 133.122,Z 372.782,A -85,B 0,C 180,E1 -25537.04,E2 -25537.04} C_VEL
LIN {X 0,Y 137.653,Z 369.721,A -85,B 0,C 180,E1 -25540.789,E2 -25540.789} C_VEL
LIN {X 0,Y 143.757,Z 364.878,A -85,B 0,C 180,E1 -25544.921,E2 -25544.921} C_VEL
LIN {X 0,Y 150.52,Z 358.604,A -85,B 0,C 180,E1 -25548.681,E2 -25548.681} C_VEL
LIN {X 0,Y 157.881,Z 350.64,A -85,B 0,C 180,E1 -25552.114,E2 -25552.114} C_VEL
LIN {X 0,Y 164.043,Z 342.854,A -85,B 0,C 180,E1 -25554.58,E2 -25554.58} C_VEL
LIN {X 0,Y 171.093,Z 332.382,A -85,B 0,C 180,E1 -25557.055,E2 -25557.055} C_VEL
LIN {X 0,Y 176.539,Z 322.74,A -85,B 0,C 180,E1 -25558.805,E2 -25558.805} C_VEL
LIN {X 0,Y 181.657,Z 311.86,A -85,B 0,C 180,E1 -25560.31,E2 -25560.31} C_VEL
LIN {X 0,Y 186.126,Z 299.709,A -85,B 0,C 180,E1 -25561.597,E2 -25561.597} C_VEL
LIN {X 0,Y 189.757,Z 286.612,A -85,B 0,C 180,E1 -25562.599,E2 -25562.599} C_VEL
LIN {X 0,Y 192.238,Z 273.624,A -85,B 0,C 180,E1 -25563.197,E2 -25563.197} C_VEL
LIN {X 0,Y 193.893,Z 259.815,A -85,B 0,C 180,E1 -25563.705,E2 -25563.705} C_VEL
LIN {X 0,Y 191.101,Z 253.091,A -85,B 0,C 180,E1 -25567.581,E2 -25567.581} C_VEL
LIN {X 0,Y 189.18,Z 249.497,A -85,B 0,C 180,E1 -25571.175,E2 -25571.175} C_VEL
LIN {X 0,Y 187.779,Z 246.457,A -85,B 0,C 180,E1 -25576.443,E2 -25576.443} C_VEL
LIN {X 0,Y 187.592,Z 246.752,A -85,B 0,C 180,E1 -25579.706,E2 -25579.706} C_VEL
LIN {X 0,Y 187.869,Z 247.785,A -85,B 0,C 180,E1 -25582.301,E2 -25582.301} C_VEL
LIN {X 0,Y 189.273,Z 252.244,A -85,B 0,C 180,E1 -25587.038,E2 -25587.038} C_VEL
LIN {X 0,Y 190.8,Z 257.08,A -85,B 0,C 180,E1 -25590.089,E2 -25590.089} C_VEL
LIN {X 0,Y 192.523,Z 262.797,A -85,B 0,C 180,E1 -25592.809,E2 -25592.809} C_VEL
LIN {X 0,Y 193.338,Z 265.725,A -85,B 0,C 180,E1 -25593.913,E2 -25593.913} C_VEL
LIN {X 0,Y 190.852,Z 284.232,A -85,B 0,C 180,E1 -25594.58,E2 -25594.58} C_VEL
LIN {X 0,Y 187.75,Z 297.722,A -85,B 0,C 180,E1 -25595.267,E2 -25595.267} C_VEL
LIN {X 0,Y 183.737,Z 309.971,A -85,B 0,C 180,E1 -25596.156,E2 -25596.156} C_VEL
LIN {X 0,Y 178.929,Z 321.485,A -85,B 0,C 180,E1 -25597.307,E2 -25597.307} C_VEL
LIN {X 0,Y 172.815,Z 333.376,A -85,B 0,C 180,E1 -25598.941,E2 -25598.941} C_VEL
LIN {X 0,Y 166.821,Z 343.005,A -85,B 0,C 180,E1 -25600.681,E2 -25600.681} C_VEL
LIN {X 0,Y 159.301,Z 353.455,A -85,B 0,C 180,E1 -25603.284,E2 -25603.284} C_VEL
LIN {X 0,Y 153.289,Z 360.583,A -85,B 0,C 180,E1 -25605.636,E2 -25605.636} C_VEL
LIN {X 0,Y 146.791,Z 367.636,A -85,B 0,C 180,E1 -25608.826,E2 -25608.826} C_VEL
LIN {X 0,Y 141.646,Z 372.476,A -85,B 0,C 180,E1 -25611.666,E2 -25611.666} C_VEL
LIN {X 0,Y 136.166,Z 377.246,A -85,B 0,C 180,E1 -25615.404,E2 -25615.404} C_VEL
LIN {X 0,Y 131.342,Z 380.993,A -85,B 0,C 180,E1 -25619.445,E2 -25619.445} C_VEL
LIN {X 0,Y 127.179,Z 383.789,A -85,B 0,C 180,E1 -25623.761,E2 -25623.761} C_VEL
LIN {X 0,Y 122.928,Z 386.15,A -85,B 0,C 180,E1 -25629.936,E2 -25629.936} C_VEL
LIN {X 0,Y 120.435,Z 386.985,A -85,B 0,C 180,E1 -25636.499,E2 -25636.499} C_VEL
LIN {X 0,Y 119.491,Z 386.315,A -85,B 0,C 180,E1 -25643.243,E2 -25643.243} C_VEL
LIN {X 0,Y 119.579,Z 385.043,A -85,B 0,C 180,E1 -25647.664,E2 -25647.664} C_VEL
LIN {X 0,Y 119.775,Z 384.092,A -85,B 0,C 180,E1 -25649.998,E2 -25649.998} C_VEL
LIN {X 0,Y 119.562,Z 381.172,A -85,B 0,C 180,E1 -25655.056,E2 -25655.056} C_VEL
LIN {X 0,Y 119.942,Z 377.143,A -85,B 0,C 180,E1 -25660.122,E2 -25660.122} C_VEL
LIN {X 0,Y 121.166,Z 370.85,A -85,B 0,C 180,E1 -25665.991,E2 -25665.991} C_VEL
LIN {X 0,Y 123.217,Z 363.977,A -85,B 0,C 180,E1 -25670.882,E2 -25670.882} C_VEL
LIN {X 0,Y 125.407,Z 356.906,A -85,B 0,C 180,E1 -25674.852,E2 -25674.852} C_VEL
LIN {X 0,Y 125.89,Z 355.405,A -85,B 0,C 180,E1 -25675.588,E2 -25675.588} C_VEL
LIN {X 0,Y 126.608,Z 351.351,A -85,B 0,C 180,E1 -25677.51,E2 -25677.51} C_VEL
LIN {X 0,Y 126.288,Z 344.248,A -85,B 0,C 180,E1 -25680.636,E2 -25680.636} C_VEL
LIN {X 0,Y 126.047,Z 336.7,A -85,B 0,C 180,E1 -25683.55,E2 -25683.55} C_VEL
LIN {X 0,Y 126.864,Z 331.828,A -85,B 0,C 180,E1 -25685.069,E2 -25685.069} C_VEL
LIN {X 0,Y 130.314,Z 320.018,A -85,B 0,C 180,E1 -25687.839,E2 -25687.839} C_VEL
LIN {X 0,Y 133.345,Z 307.57,A -85,B 0,C 180,E1 -25689.965,E2 -25689.965} C_VEL
LIN {X 0,Y 135.71,Z 294.599,A -85,B 0,C 180,E1 -25691.567,E2 -25691.567} C_VEL
LIN {X 0,Y 137.42,Z 281.549,A -85,B 0,C 180,E1 -25692.583,E2 -25692.583} C_VEL
LIN {X 0,Y 140.141,Z 244.207,A -85,B 0,C 180,E1 -25694.576,E2 -25694.576} C_VEL
LIN {X 0,Y 139.147,Z 231.597,A -85,B 0,C 180,E1 -25695.743,E2 -25695.743} C_VEL
LIN {X 0,Y 133.15,Z 214.189,A -85,B 0,C 180,E1 -25698.832,E2 -25698.832} C_VEL
LIN {X 0,Y 127.175,Z 200.077,A -85,B 0,C 180,E1 -25702.022,E2 -25702.022} C_VEL
LIN {X 0,Y 124.025,Z 194.396,A -85,B 0,C 180,E1 -25703.709,E2 -25703.709} C_VEL
LIN {X 0,Y 119.622,Z 187.387,A -85,B 0,C 180,E1 -25706.197,E2 -25706.197} C_VEL
LIN {X 0,Y 117.395,Z 183.771,A -85,B 0,C 180,E1 -25707.56,E2 -25707.56} C_VEL
LIN {X 0,Y 115.523,Z 181.373,A -85,B 0,C 180,E1 -25708.706,E2 -25708.706} C_VEL
LIN {X 0,Y 114.891,Z 179.167,A -85,B 0,C 180,E1 -25709.346,E2 -25709.346} C_VEL
LIN {X 0,Y 114.945,Z 179.155,A -85,B 0,C 180,E1 -25716.506,E2 -25716.506} C_VEL
LIN {X 0,Y 114.988,Z 179.151,A -85,B 0,C 180,E1 -25722.204,E2 -25722.204} C_VEL
LIN {X 0,Y 115.261,Z 179.129,A -85,B 0,C 180,E1 -25727.306,E2 -25727.306} C_VEL
LIN {X 0,Y 115.386,Z 179.092,A -85,B 0,C 180,E1 -25733.001,E2 -25733.001} C_VEL
LIN {X 0,Y 115.993,Z 179.022,A -85,B 0,C 180,E1 -25739.998,E2 -25739.998} C_VEL
LIN {X 0,Y 115.385,Z 179.111,A -85,B 0,C 180,E1 -25747.009,E2 -25747.009} C_VEL
LIN {X 0,Y 115.281,Z 179.099,A -85,B 0,C 180,E1 -25752.736,E2 -25752.736} C_VEL
LIN {X 0,Y 115.015,Z 179.153,A -85,B 0,C 180,E1 -25757.788,E2 -25757.788} C_VEL
LIN {X 0,Y 114.942,Z 179.144,A -85,B 0,C 180,E1 -25763.491,E2 -25763.491} C_VEL
LIN {X 0,Y 114.865,Z 179.171,A -85,B 0,C 180,E1 -25771.068,E2 -25771.068} C_VEL
LIN {X 0,Y 114.877,Z 179.151,A -85,B 0,C 180,E1 -25777.716,E2 -25777.716} C_VEL
LIN {X 0,Y 114.883,Z 179.168,A -85,B 0,C 180,E1 -25782.772,E2 -25782.772} C_VEL
LIN {X 0,Y 114.89,Z 179.158,A -85,B 0,C 180,E1 -25787.712,E2 -25787.712} C_VEL
LIN {X 0,Y 114.89,Z 179.166,A -85,B 0,C 180,E1 -25792.673,E2 -25792.673} C_VEL
LIN {X 0,Y 114.865,Z 179.177,A -85,B 0,C 180,E1 -25798.931,E2 -25798.931} C_VEL
LIN {X 0,Y 114.942,Z 179.166,A -85,B 0,C 180,E1 -25806.509,E2 -25806.509} C_VEL
LIN {X 0,Y 115.025,Z 179.309,A -85,B 0,C 180,E1 -25809.696,E2 -25809.696} C_VEL
LIN {X 0,Y 115.957,Z 181.925,A -85,B 0,C 180,E1 -25810.423,E2 -25810.423} C_VEL
LIN {X 0,Y 118.121,Z 184.527,A -85,B 0,C 180,E1 -25811.696,E2 -25811.696} C_VEL
LIN {X 0,Y 120.374,Z 187.938,A -85,B 0,C 180,E1 -25813.029,E2 -25813.029} C_VEL
LIN {X 0,Y 125.636,Z 196.039,A -85,B 0,C 180,E1 -25815.924,E2 -25815.924} C_VEL
LIN {X 0,Y 134.692,Z 212.368,A -85,B 0,C 180,E1 -25820.364,E2 -25820.364} C_VEL
LIN {X 0,Y 141.131,Z 227.787,A -85,B 0,C 180,E1 -25823.379,E2 -25823.379} C_VEL
LIN {X 0,Y 137.506,Z 273.26,A -85,B 0,C 180,E1 -25825.752,E2 -25825.752} C_VEL
LIN {X 0,Y 135.737,Z 286.719,A -85,B 0,C 180,E1 -25826.976,E2 -25826.976} C_VEL
LIN {X 0,Y 133.565,Z 299.079,A -85,B 0,C 180,E1 -25828.647,E2 -25828.647} C_VEL
LIN {X 0,Y 130.94,Z 310.606,A -85,B 0,C 180,E1 -25830.771,E2 -25830.771} C_VEL
LIN {X 0,Y 127.473,Z 322.757,A -85,B 0,C 180,E1 -25833.723,E2 -25833.723} C_VEL
LIN {X 0,Y 123.905,Z 333.908,A -85,B 0,C 180,E1 -25837.334,E2 -25837.334} C_VEL
LIN {X 0,Y 120.651,Z 343.434,A -85,B 0,C 180,E1 -25841.378,E2 -25841.378} C_VEL
LIN {X 0,Y 118.013,Z 351.144,A -85,B 0,C 180,E1 -25845.547,E2 -25845.547} C_VEL
LIN {X 0,Y 115.575,Z 358.34,A -85,B 0,C 180,E1 -25850.468,E2 -25850.468} C_VEL
LIN {X 0,Y 113.816,Z 364.191,A -85,B 0,C 180,E1 -25855.612,E2 -25855.612} C_VEL
LIN {X 0,Y 112.344,Z 369.735,A -85,B 0,C 180,E1 -25862.126,E2 -25862.126} C_VEL
LIN {X 0,Y 111.948,Z 373.787,A -85,B 0,C 180,E1 -25868.89,E2 -25868.89} C_VEL
LIN {X 0,Y 112.403,Z 375.632,A -85,B 0,C 180,E1 -25873.457,E2 -25873.457} C_VEL
LIN {X 0,Y 113.437,Z 376.885,A -85,B 0,C 180,E1 -25878.03,E2 -25878.03} C_VEL
LIN {X 0,Y 115.075,Z 377.459,A -85,B 0,C 180,E1 -25882.56,E2 -25882.56} C_VEL
LIN {X 0,Y 117.597,Z 377.347,A -85,B 0,C 180,E1 -25887.464,E2 -25887.464} C_VEL
LIN {X 0,Y 120.964,Z 376.389,A -85,B 0,C 180,E1 -25892.305,E2 -25892.305} C_VEL
LIN {X 0,Y 125.147,Z 374.558,A -85,B 0,C 180,E1 -25896.854,E2 -25896.854} C_VEL
LIN {X 0,Y 130.023,Z 371.819,A -85,B 0,C 180,E1 -25901.078,E2 -25901.078} C_VEL
LIN {X 0,Y 135.496,Z 368.107,A -85,B 0,C 180,E1 -25904.971,E2 -25904.971} C_VEL
LIN {X 0,Y 143.037,Z 362.009,A -85,B 0,C 180,E1 -25909.331,E2 -25909.331} C_VEL
LIN {X 0,Y 150.518,Z 354.905,A -85,B 0,C 180,E1 -25912.856,E2 -25912.856} C_VEL
LIN {X 0,Y 156.867,Z 347.864,A -85,B 0,C 180,E1 -25915.47,E2 -25915.47} C_VEL
LIN {X 0,Y 163.687,Z 339.189,A -85,B 0,C 180,E1 -25917.836,E2 -25917.836} C_VEL
LIN {X 0,Y 170.496,Z 328.745,A -85,B 0,C 180,E1 -25920.001,E2 -25920.001} C_VEL
LIN {X 0,Y 176.606,Z 317.415,A -85,B 0,C 180,E1 -25921.754,E2 -25921.754} C_VEL
LIN {X 0,Y 181.654,Z 305.594,A -85,B 0,C 180,E1 -25923.124,E2 -25923.124} C_VEL
LIN {X 0,Y 185.69,Z 293.43,A -85,B 0,C 180,E1 -25924.176,E2 -25924.176} C_VEL
LIN {X 0,Y 188.414,Z 282.44,A -85,B 0,C 180,E1 -25924.86,E2 -25924.86} C_VEL
LIN {X 0,Y 190.692,Z 268.53,A -85,B 0,C 180,E1 -25925.411,E2 -25925.411} C_VEL
LIN {X 0,Y 191.186,Z 264.187,A -85,B 0,C 180,E1 -25925.596,E2 -25925.596} C_VEL
LIN {X 0,Y 189.483,Z 259.573,A -85,B 0,C 180,E1 -25928.345,E2 -25928.345} C_VEL
LIN {X 0,Y 187.853,Z 256.288,A -85,B 0,C 180,E1 -25931.743,E2 -25931.743} C_VEL
LIN {X 0,Y 186.713,Z 253.472,A -85,B 0,C 180,E1 -25936.539,E2 -25936.539} C_VEL
LIN {X 0,Y 186.546,Z 253.809,A -85,B 0,C 180,E1 -25939.821,E2 -25939.821} C_VEL
LIN {X 0,Y 186.735,Z 254.651,A -85,B 0,C 180,E1 -25941.844,E2 -25941.844} C_VEL
LIN {X 0,Y 187.909,Z 258.996,A -85,B 0,C 180,E1 -25946.442,E2 -25946.442} C_VEL
LIN {X 0,Y 189.092,Z 263.318,A -85,B 0,C 180,E1 -25949.182,E2 -25949.182} C_VEL
LIN {X 0,Y 190.405,Z 268.105,A -85,B 0,C 180,E1 -25951.54,E2 -25951.54} C_VEL
LIN {X 0,Y 190.686,Z 269.37,A -85,B 0,C 180,E1 -25952.035,E2 -25952.035} C_VEL
LIN {X 0,Y 188.329,Z 285.209,A -85,B 0,C 180,E1 -25952.602,E2 -25952.602} C_VEL
LIN {X 0,Y 184.958,Z 298.736,A -85,B 0,C 180,E1 -25953.282,E2 -25953.282} C_VEL
LIN {X 0,Y 180.561,Z 311.403,A -85,B 0,C 180,E1 -25954.194,E2 -25954.194} C_VEL
LIN {X 0,Y 175.522,Z 322.772,A -85,B 0,C 180,E1 -25955.329,E2 -25955.329} C_VEL
LIN {X 0,Y 169.219,Z 334.276,A -85,B 0,C 180,E1 -25956.916,E2 -25956.916} C_VEL
LIN {X 0,Y 162.367,Z 344.635,A -85,B 0,C 180,E1 -25958.817,E2 -25958.817} C_VEL
LIN {X 0,Y 155.855,Z 353.114,A -85,B 0,C 180,E1 -25960.945,E2 -25960.945} C_VEL
LIN {X 0,Y 148.336,Z 361.483,A -85,B 0,C 180,E1 -25963.734,E2 -25963.734} C_VEL
LIN {X 0,Y 141.543,Z 368.284,A -85,B 0,C 180,E1 -25966.941,E2 -25966.941} C_VEL
LIN {X 0,Y 134.126,Z 374.635,A -85,B 0,C 180,E1 -25971.038,E2 -25971.038} C_VEL
LIN {X 0,Y 127.999,Z 379.298,A -85,B 0,C 180,E1 -25975.45,E2 -25975.45} C_VEL
LIN {X 0,Y 123.727,Z 382.113,A -85,B 0,C 180,E1 -25979.252,E2 -25979.252} C_VEL
LIN {X 0,Y 118.392,Z 385.079,A -85,B 0,C 180,E1 -25985.445,E2 -25985.445} C_VEL
LIN {X 0,Y 114.641,Z 386.472,A -85,B 0,C 180,E1 -25992.148,E2 -25992.148} C_VEL
LIN {X 0,Y 112.786,Z 386.402,A -85,B 0,C 180,E1 -25999.224,E2 -25999.224} C_VEL
LIN {X 0,Y 112.432,Z 385.818,A -85,B 0,C 180,E1 -26002.816,E2 -26002.816} C_VEL
LIN {X 0,Y 112.534,Z 384.311,A -85,B 0,C 180,E1 -26007.805,E2 -26007.805} C_VEL
LIN {X 0,Y 112.708,Z 383.396,A -85,B 0,C 180,E1 -26009.998,E2 -26009.998} C_VEL
LIN {X 0,Y 112.505,Z 380.331,A -85,B 0,C 180,E1 -26015.375,E2 -26015.375} C_VEL
LIN {X 0,Y 112.947,Z 376.145,A -85,B 0,C 180,E1 -26020.756,E2 -26020.756} C_VEL
LIN {X 0,Y 114.328,Z 369.681,A -85,B 0,C 180,E1 -26026.975,E2 -26026.975} C_VEL
LIN {X 0,Y 116.579,Z 362.587,A -85,B 0,C 180,E1 -26032.132,E2 -26032.132} C_VEL
LIN {X 0,Y 119.517,Z 353.635,A -85,B 0,C 180,E1 -26037.11,E2 -26037.11} C_VEL
LIN {X 0,Y 122.759,Z 344.5,A -85,B 0,C 180,E1 -26041.012,E2 -26041.012} C_VEL
LIN {X 0,Y 126.133,Z 334.406,A -85,B 0,C 180,E1 -26044.341,E2 -26044.341} C_VEL
LIN {X 0,Y 126.864,Z 331.828,A -85,B 0,C 180,E1 -26045.069,E2 -26045.069} C_VEL
LIN {X 0,Y 127.683,Z 326.882,A -85,B 0,C 180,E1 -26046.486,E2 -26046.486} C_VEL
LIN {X 0,Y 127.497,Z 318.499,A -85,B 0,C 180,E1 -26048.87,E2 -26048.87} C_VEL
LIN {X 0,Y 127.188,Z 309.755,A -85,B 0,C 180,E1 -26050.978,E2 -26050.978} C_VEL
LIN {X 0,Y 127.768,Z 304.244,A -85,B 0,C 180,E1 -26051.915,E2 -26051.915} C_VEL
LIN {X 0,Y 130.218,Z 290.38,A -85,B 0,C 180,E1 -26053.48,E2 -26053.48} C_VEL
LIN {X 0,Y 131.708,Z 277.579,A -85,B 0,C 180,E1 -26054.386,E2 -26054.386} C_VEL
LIN {X 0,Y 134.158,Z 245.058,A -85,B 0,C 180,E1 -26056.151,E2 -26056.151} C_VEL
LIN {X 0,Y 133.326,Z 233.843,A -85,B 0,C 180,E1 -26057.25,E2 -26057.25} C_VEL
LIN {X 0,Y 128.005,Z 217.943,A -85,B 0,C 180,E1 -26060.236,E2 -26060.236} C_VEL
LIN {X 0,Y 122.343,Z 204.135,A -85,B 0,C 180,E1 -26063.502,E2 -26063.502} C_VEL
LIN {X 0,Y 119.011,Z 198.07,A -85,B 0,C 180,E1 -26065.456,E2 -26065.456} C_VEL
LIN {X 0,Y 113.43,Z 189.105,A -85,B 0,C 180,E1 -26068.953,E2 -26068.953} C_VEL
LIN {X 0,Y 111.251,Z 185.899,A -85,B 0,C 180,E1 -26070.425,E2 -26070.425} C_VEL
LIN {X 0,Y 110.47,Z 184.722,A -85,B 0,C 180,E1 -26070.979,E2 -26070.979} C_VEL
LIN {X 0,Y 108.603,Z 182.614,A -85,B 0,C 180,E1 -26072.28,E2 -26072.28} C_VEL
LIN {X 0,Y 107.777,Z 180.061,A -85,B 0,C 180,E1 -26073.187,E2 -26073.187} C_VEL
LIN {X 0,Y 107.906,Z 180.032,A -85,B 0,C 180,E1 -26076.995,E2 -26076.995} C_VEL
LIN {X 0,Y 108.021,Z 180.017,A -85,B 0,C 180,E1 -26084.913,E2 -26084.913} C_VEL
LIN {X 0,Y 108.273,Z 179.996,A -85,B 0,C 180,E1 -26088.769,E2 -26088.769} C_VEL
LIN {X 0,Y 108.456,Z 179.973,A -85,B 0,C 180,E1 -26096.283,E2 -26096.283} C_VEL
LIN {X 0,Y 108.943,Z 179.9,A -85,B 0,C 180,E1 -26099.998,E2 -26099.998} C_VEL
LIN {X 0,Y 108.326,Z 179.991,A -85,B 0,C 180,E1 -26107.453,E2 -26107.453} C_VEL
LIN {X 0,Y 108.195,Z 179.979,A -85,B 0,C 180,E1 -26113.015,E2 -26113.015} C_VEL
LIN {X 0,Y 107.905,Z 180.042,A -85,B 0,C 180,E1 -26119.003,E2 -26119.003} C_VEL
LIN {X 0,Y 107.853,Z 180.021,A -85,B 0,C 180,E1 -26124.183,E2 -26124.183} C_VEL
LIN {X 0,Y 107.796,Z 180.05,A -85,B 0,C 180,E1 -26132.056,E2 -26132.056} C_VEL
LIN {X 0,Y 107.781,Z 180.04,A -85,B 0,C 180,E1 -26138.516,E2 -26138.516} C_VEL
LIN {X 0,Y 107.783,Z 180.036,A -85,B 0,C 180,E1 -26145.825,E2 -26145.825} C_VEL
LIN {X 0,Y 107.787,Z 180.056,A -85,B 0,C 180,E1 -26151.48,E2 -26151.48} C_VEL
LIN {X 0,Y 107.807,Z 180.056,A -85,B 0,C 180,E1 -26158.568,E2 -26158.568} C_VEL
LIN {X 0,Y 107.871,Z 180.048,A -85,B 0,C 180,E1 -26165.796,E2 -26165.796} C_VEL
LIN {X 0,Y 108.919,Z 182.922,A -85,B 0,C 180,E1 -26166.799,E2 -26166.799} C_VEL
LIN {X 0,Y 111.148,Z 185.362,A -85,B 0,C 180,E1 -26168.328,E2 -26168.328} C_VEL
LIN {X 0,Y 113.233,Z 188.714,A -85,B 0,C 180,E1 -26169.781,E2 -26169.781} C_VEL
LIN {X 0,Y 117.419,Z 194.932,A -85,B 0,C 180,E1 -26172.396,E2 -26172.396} C_VEL
LIN {X 0,Y 122.073,Z 202.269,A -85,B 0,C 180,E1 -26175.077,E2 -26175.077} C_VEL
LIN {X 0,Y 130.158,Z 217.545,A -85,B 0,C 180,E1 -26179.316,E2 -26179.316} C_VEL
LIN {X 0,Y 135.052,Z 229.639,A -85,B 0,C 180,E1 -26181.796,E2 -26181.796} C_VEL
LIN {X 0,Y 131.494,Z 273.28,A -85,B 0,C 180,E1 -26184.154,E2 -26184.154} C_VEL
LIN {X 0,Y 129.602,Z 287.029,A -85,B 0,C 180,E1 -26185.434,E2 -26185.434} C_VEL
LIN {X 0,Y 127.317,Z 299.473,A -85,B 0,C 180,E1 -26187.174,E2 -26187.174} C_VEL
LIN {X 0,Y 124.587,Z 310.935,A -85,B 0,C 180,E1 -26189.365,E2 -26189.365} C_VEL
LIN {X 0,Y 120.894,Z 323.322,A -85,B 0,C 180,E1 -26192.501,E2 -26192.501} C_VEL
LIN {X 0,Y 117.378,Z 333.782,A -85,B 0,C 180,E1 -26196.022,E2 -26196.022} C_VEL
LIN {X 0,Y 114.165,Z 342.78,A -85,B 0,C 180,E1 -26199.961,E2 -26199.961} C_VEL
LIN {X 0,Y 111.164,Z 351.124,A -85,B 0,C 180,E1 -26204.651,E2 -26204.651} C_VEL
LIN {X 0,Y 108.572,Z 358.374,A -85,B 0,C 180,E1 -26209.869,E2 -26209.869} C_VEL
LIN {X 0,Y 106.704,Z 364.319,A -85,B 0,C 180,E1 -26215.385,E2 -26215.385} C_VEL
LIN {X 0,Y 105.21,Z 369.886,A -85,B 0,C 180,E1 -26222.306,E2 -26222.306} C_VEL
LIN {X 0,Y 104.874,Z 373.999,A -85,B 0,C 180,E1 -26229.544,E2 -26229.544} C_VEL
LIN {X 0,Y 105.94,Z 376.622,A -85,B 0,C 180,E1 -26236.868,E2 -26236.868} C_VEL
LIN {X 0,Y 108.631,Z 377.816,A -85,B 0,C 180,E1 -26244.393,E2 -26244.393} C_VEL
LIN {X 0,Y 112.471,Z 377.535,A -85,B 0,C 180,E1 -26251.028,E2 -26251.028} C_VEL
LIN {X 0,Y 115.969,Z 376.488,A -85,B 0,C 180,E1 -26255.377,E2 -26255.377} C_VEL
LIN {X 0,Y 122.353,Z 373.677,A -85,B 0,C 180,E1 -26261.406,E2 -26261.406} C_VEL
LIN {X 0,Y 127.423,Z 370.765,A -85,B 0,C 180,E1 -26265.178,E2 -26265.178} C_VEL
LIN {X 0,Y 133.197,Z 366.879,A -85,B 0,C 180,E1 -26268.747,E2 -26268.747} C_VEL
LIN {X 0,Y 139.449,Z 362.044,A -85,B 0,C 180,E1 -26271.98,E2 -26271.98} C_VEL
LIN {X 0,Y 146.147,Z 356.037,A -85,B 0,C 180,E1 -26274.973,E2 -26274.973} C_VEL
LIN {X 0,Y 153.128,Z 348.76,A -85,B 0,C 180,E1 -26277.682,E2 -26277.682} C_VEL
